// TwinCAT 3 PLC project ModbusExt2
// Title: ModbusExt2
// Company: Beckhoff Automation
// ProjectVersion: 0.1.0.0
// ProgramVersion: 3.1.4026.27
// libraries:
//   Tc2_SerialCom, * (Beckhoff Automation GmbH)
//   Tc2_Standard, * (Beckhoff Automation GmbH)
//   Tc2_System, * (Beckhoff Automation GmbH)
//   Tc2_TcpIp, * (Beckhoff Automation GmbH)
//   Tc2_Utilities, * (Beckhoff Automation GmbH)
// project tree:
//   DUTs/ E_MbAddressing.TcDUT, E_MbDevState.TcDUT, E_MbErrorClass.TcDUT, E_MbLogWriterStep.TcDUT, E_MbOp.TcDUT, E_MbPoll.TcDUT, E_MbRegion.TcDUT, E_MbTcpConn.TcDUT, E_MbType.TcDUT, E_MbWordOrder.TcDUT, E_MbXferState.TcDUT, ST_MbBlock.TcDUT, ST_MbLog.TcDUT, ST_MbLogEntry.TcDUT, ST_MbParseResult.TcDUT, ST_MbPoint.TcDUT, ST_MbPointState.TcDUT, ST_MbProbe.TcDUT, ST_MbProfile.TcDUT, U_MbConv.TcDUT
//   GVLs/ GVL_MbConst.TcGVL, GVL_MbParam.TcGVL
//   POUs/Codec/ F_MbCrc16.TcPOU, F_MbDecode.TcPOU, F_MbEncode.TcPOU, F_MbExpectedResponseLength.TcPOU, F_MbBuildRequest.TcPOU, F_MbMemCpy.TcPOU, F_MbMemSet.TcPOU, F_MbParseResponse.TcPOU, F_MbRound.TcPOU, F_MbTimeToFt.TcPOU
//   POUs/Device/ FB_ModbusDevice.TcPOU
//   POUs/Log/ FB_MbLogExport.TcPOU, FB_MbLogWriter.TcPOU, F_MbLogEntryToCsv.TcPOU
//   POUs/Profiles/ FB_Mb_CorrAll.TcPOU
//   POUs/Transport/ FB_MbTransportMock.TcPOU, FB_MbTransportRtu.TcPOU, FB_MbTransportTcp.TcPOU, I_MbTransport.TcIO
// real-time tasks:
//   TASK PlcTask1: cycle T#10ms, priority 21, ADS port 351
//   TASK PlcTask: cycle T#10ms, priority 20, ADS port 350

// ---- DUTs/E_MbAddressing.TcDUT
{attribute 'qualified_only'}
{attribute 'strict'}
TYPE E_MbAddressing :
(
	Modicon := 0,
	Offset0,
	Offset1
);
END_TYPE

// ---- DUTs/E_MbDevState.TcDUT
{attribute 'qualified_only'}
{attribute 'strict'}
TYPE E_MbDevState :
(
	Idle := 0,
	Acquire,
	Wait,
	Cooldown
);
END_TYPE

// ---- DUTs/E_MbErrorClass.TcDUT
{attribute 'qualified_only'}
{attribute 'strict'}
{attribute 'to_string'}
TYPE E_MbErrorClass :
(
	None := 0,
	Timeout,
	Crc,
	Exception,
	Transport,
	Config,
	Truncated,
	Malformed,
	StillFailing,
	Recovered
);
END_TYPE

// ---- DUTs/E_MbLogWriterStep.TcDUT
{attribute 'qualified_only'}
{attribute 'strict'}
TYPE E_MbLogWriterStep :
(
	Idle := 0,
	MkDir,
	MkDirWait,
	Open,
	OpenWait,
	SeekWait,
	TellWait,
	PutWait,
	CloseWait,
	DeleteWait,
	RenameWait
);
END_TYPE

// ---- DUTs/E_MbOp.TcDUT
{attribute 'qualified_only'}
{attribute 'strict'}
{attribute 'to_string'}
TYPE E_MbOp :
(
	Read := 0,
	Write
);
END_TYPE

// ---- DUTs/E_MbPoll.TcDUT
{attribute 'qualified_only'}
{attribute 'strict'}
TYPE E_MbPoll :
(
	Fast := 0,
	Slow,
	Off
);
END_TYPE

// ---- DUTs/E_MbRegion.TcDUT
{attribute 'qualified_only'}
{attribute 'strict'}
{attribute 'to_string'}
TYPE E_MbRegion :
(
	Auto := 0,
	Coil,
	DiscreteInput,
	InputRegister,
	HoldingRegister
);
END_TYPE

// ---- DUTs/E_MbTcpConn.TcDUT
{attribute 'qualified_only'}
{attribute 'strict'}
TYPE E_MbTcpConn :
(
	Init := 0,
	CloseAllWait,
	Disconnected,
	Connecting,
	Connected,
	Closing,
	ClosingWait
);
END_TYPE

// ---- DUTs/E_MbType.TcDUT
{attribute 'qualified_only'}
{attribute 'strict'}
TYPE E_MbType :
(
	Auto := 0,
	Boolean,
	Int16,
	UInt16,
	Int32,
	UInt32,
	Real32,
	Int64,
	UInt64,
	Real64,
	RegisterBit,
	Text,
	Raw
);
END_TYPE

// ---- DUTs/E_MbWordOrder.TcDUT
{attribute 'qualified_only'}
{attribute 'strict'}
TYPE E_MbWordOrder :
(
	Inherit := 0,
	ABCD,
	CDAB,
	BADC,
	DCBA
);
END_TYPE

// ---- DUTs/E_MbXferState.TcDUT
{attribute 'qualified_only'}
{attribute 'strict'}
TYPE E_MbXferState :
(
	Idle := 0,
	Busy,
	Done,
	Timeout,
	Error
);
END_TYPE

// ---- DUTs/ST_MbBlock.TcDUT
TYPE ST_MbBlock :
STRUCT
	eRegion      : E_MbRegion;
	nOffset      : UINT;       // 0-based start address
	nCount       : UINT;       // Registers or coils
	nFc          : USINT;      // Read function code
	ePoll        : E_MbPoll;
	nSortedFirst : UINT;       // Index range into FB_ModbusDevice.aSorted
	nSortedCount : UINT;
	tLastPoll    : ULINT;      // FILETIME of last completed poll (Slow scheduling)
	nConsecFail  : UINT;
END_STRUCT
END_TYPE

// ---- DUTs/ST_MbLog.TcDUT
TYPE ST_MbLog :
STRUCT
	aEntries     : ARRAY[0..GVL_MbParam.MB_LOG_SIZE-1] OF ST_MbLogEntry;
	nHead        : UINT;                             // Next write index
	nCount       : UINT;                             // Valid entries, <= MB_LOG_SIZE
	nTotalErrors : UDINT;
	nDropped     : UDINT;                            // Entries overwritten by ring wrap
	nSeq         : UDINT;                            // Entries ever written; the file writer's cursor
END_STRUCT
END_TYPE

// ---- DUTs/ST_MbLogEntry.TcDUT
TYPE ST_MbLogEntry :
STRUCT
	tTime    : ULINT;                                // FILETIME (100 ns, UTC)
	sName    : STRING(GVL_MbParam.MB_NAME_LEN);
	nUnitId  : USINT;
	eRegion  : E_MbRegion;
	nAddr    : UDINT;                                // As entered in the profile
	nFc      : BYTE;
	eOp      : E_MbOp;
	eClass   : E_MbErrorClass;
	nExcCode : BYTE;
	nRetries : USINT;
	nRepeat  : UDINT;                                // StillFailing: occurrences since first failure
END_STRUCT
END_TYPE

// ---- DUTs/ST_MbParseResult.TcDUT
TYPE ST_MbParseResult :
STRUCT
	bOk         : BOOL;             // Valid non-exception response matching the request
	bException  : BOOL;
	nExcCode    : BYTE;             // Modbus exception code when bException
	eClass      : E_MbErrorClass;   // None | Exception | Truncated | Malformed
	nByteCount  : UINT;             // Data bytes (FC 1..4)
	nDataOffset : UINT;             // Index of first data byte within the PDU (FC 1..4)
END_STRUCT
END_TYPE

// ---- DUTs/ST_MbPoint.TcDUT
TYPE ST_MbPoint :
STRUCT
	// ---- Profile fills these ----
	nAddr         : UDINT;                                   // Address as printed in the device manual (see E_MbAddressing)
	eType         : E_MbType     := E_MbType.Auto;           // Auto: Boolean for bit regions, UInt16 for registers
	eRegion       : E_MbRegion   := E_MbRegion.Auto;         // Auto: derived from nAddr (Modicon); required for Offset0/Offset1
	eWordOrder    : E_MbWordOrder := E_MbWordOrder.Inherit;  // Inherit from Profile()
	fRawMin       : LREAL;                                   // Scaling active iff fRawMin <> fRawMax
	fRawMax       : LREAL;
	fEngMin       : LREAL;
	fEngMax       : LREAL;
	fGain         : LREAL;                                   // Alternative scaling: eng = raw * fGain + fOffset. Active iff fGain <> 0
	fOffset       : LREAL;
	ePoll         : E_MbPoll     := E_MbPoll.Fast;
	bUseFailValue : BOOL;                                    // TRUE: fValue := fFailValue after retries exhausted
	fFailValue    : LREAL;
	nRegs         : UINT;                                    // Text/Raw only: registers to read
	nBit          : USINT;                                   // RegisterBit only: 0..15

	// ---- Library fills these ----
	fValue        : LREAL;                                   // Scaled value (numeric, Boolean, RegisterBit)
	sValue        : STRING(GVL_MbParam.MB_STR_LEN);          // Text
	aRaw          : ARRAY[0..GVL_MbParam.MB_RAW_WORDS-1] OF WORD;  // Raw, and raw words of every read
	bValid        : BOOL;
	tLastGood     : ULINT;                                   // FILETIME (100 ns, UTC) of last good read
	nFailCount    : UDINT;
	bProbe        : BOOL;                                    // User sets; cleared after stProbe is filled

	// ---- Write handshake ----
	fWriteValue   : LREAL;
	bWriteReq     : BOOL;
	bWriteBusy    : BOOL;
	bWriteDone    : BOOL;
	bWriteErr     : BOOL;

	// ---- Internal ----
	wMagic        : WORD := 16#4D50;
	nIndex        : UINT;
END_STRUCT
END_TYPE

// ---- DUTs/ST_MbPointState.TcDUT
TYPE ST_MbPointState :
STRUCT
	pPoint      : POINTER TO ST_MbPoint;   // Re-established in FB_reinit
	sName       : STRING(GVL_MbParam.MB_NAME_LEN);
	eRegion     : E_MbRegion;              // Resolved
	nOffset     : UINT;                    // Resolved 0-based address
	nCount      : UINT;                    // Registers or coils occupied
	eType       : E_MbType;                // Resolved (Auto replaced)
	eWordOrder  : E_MbWordOrder;           // Resolved (Inherit replaced)
	nReadFc     : USINT;
	nWriteFc    : USINT;                   // 0 = not writable
	nBlock      : UINT;                    // Owning read block; MB_MAX_BLOCKS = none (Poll Off)
	bFailing    : BOOL;
	nRepeat     : UDINT;
	tLastLog    : ULINT;
	eLastClass  : E_MbErrorClass;
	nLastExc    : BYTE;
	nWriteState : USINT;                   // 0 idle, 1 queued, 2 in flight
	aWriteData  : ARRAY[0..7] OF BYTE;
	cbWriteData : USINT;
	nWriteQty   : UINT;
END_STRUCT
END_TYPE

// ---- DUTs/ST_MbProbe.TcDUT
TYPE ST_MbProbe :
STRUCT
	sName        : STRING(GVL_MbParam.MB_NAME_LEN);
	nAddr        : UDINT;
	aRaw         : ARRAY[0..3] OF WORD;              // First four registers as received
	nInt16       : INT;
	nUInt16      : UINT;
	nInt32_ABCD  : DINT;
	nInt32_CDAB  : DINT;
	nInt32_BADC  : DINT;
	nInt32_DCBA  : DINT;
	nUInt32_ABCD : UDINT;
	nUInt32_CDAB : UDINT;
	nUInt32_BADC : UDINT;
	nUInt32_DCBA : UDINT;
	fReal32_ABCD : REAL;
	fReal32_CDAB : REAL;
	fReal32_BADC : REAL;
	fReal32_DCBA : REAL;
END_STRUCT
END_TYPE

// ---- DUTs/ST_MbProfile.TcDUT
TYPE ST_MbProfile :
STRUCT
	sModel          : STRING(GVL_MbParam.MB_NAME_LEN);
	eWordOrder      : E_MbWordOrder  := E_MbWordOrder.ABCD;
	eAddressing     : E_MbAddressing := E_MbAddressing.Modicon;
	nMaxRegsPerRead : UINT := GVL_MbConst.MAX_READ_REGS;
	nMaxGap         : UINT := 8;
	bFc6Only        : BOOL;
	bFc16Only       : BOOL;
	bStringByteSwap : BOOL;
	tSlowPoll       : TIME := T#5S;
END_STRUCT
END_TYPE

// ---- DUTs/U_MbConv.TcDUT
TYPE U_MbConv :
UNION
	lw : LWORD;
	dw : DWORD;
	w  : WORD;
	i  : INT;
	di : DINT;
	li : LINT;
	fR : REAL;
	fL : LREAL;
END_UNION
END_TYPE

// ---- GVLs/GVL_MbConst.TcGVL
{attribute 'qualified_only'}
VAR_GLOBAL CONSTANT
	FC_READ_COILS      : USINT := 1;
	FC_READ_DISCRETE   : USINT := 2;
	FC_READ_HOLDING    : USINT := 3;
	FC_READ_INPUT      : USINT := 4;
	FC_WRITE_COIL      : USINT := 5;
	FC_WRITE_REGISTER  : USINT := 6;
	FC_WRITE_COILS     : USINT := 15;
	FC_WRITE_REGISTERS : USINT := 16;
	EXC_FLAG           : BYTE  := 16#80;
	MAX_READ_REGS      : UINT  := 125;
	MAX_WRITE_REGS     : UINT  := 123;
	MAX_READ_COILS     : UINT  := 2000;
	MAX_WRITE_COILS    : UINT  := 1968;
	CFG_TOO_MANY_POINTS : BYTE := 1;
	CFG_NO_POINTS       : BYTE := 2;
	CFG_BAD_MAGIC       : BYTE := 3;
	CFG_EMPTY_NAME      : BYTE := 4;
	CFG_DUP_NAME        : BYTE := 5;
	CFG_BAD_ADDRESS     : BYTE := 6;
	CFG_REGION_REQUIRED : BYTE := 7;
	CFG_REGION_MISMATCH : BYTE := 8;
	CFG_BAD_TYPE        : BYTE := 9;
	CFG_BAD_REGS        : BYTE := 10;
	CFG_BAD_BIT         : BYTE := 11;
	CFG_BAD_SCALING     : BYTE := 12;
	CFG_OVERLAP         : BYTE := 13;
	CFG_TOO_MANY_BLOCKS : BYTE := 14;
	CFG_BAD_FAILVALUE   : BYTE := 15;
	CFG_NO_TRANSPORT    : BYTE := 16;
	CFG_NOT_WRITABLE    : BYTE := 17;
	CFG_WRITE_RANGE     : BYTE := 18;
END_VAR

// ---- GVLs/GVL_MbParam.TcGVL
{attribute 'qualified_only'}
VAR_GLOBAL CONSTANT
	MB_MAX_POINTS                : UINT := 256;
	MB_MAX_BLOCKS                : UINT := 64;
	MB_LOG_SIZE                  : UINT := 100;
	MB_STR_LEN                   : UINT := 32;
	MB_RAW_WORDS                 : UINT := 8;
	MB_NAME_LEN                  : UINT := 32;
	MB_MAX_DEVICES_PER_TRANSPORT : UINT := 32;
	MB_ADU_SIZE                  : UINT := 260;
	MB_LOG_REPEAT_INTERVAL       : TIME := T#5M;
	MB_OFFLINE_RETRY             : TIME := T#5S;
	MB_LOG_DIR                   : STRING(255) := 'C:\ModbusExt\Logs\';
	MB_LOG_FILE_MAX_BYTES        : UDINT := 2000000;   // Rotate to <name>.1.csv above this
	MB_LOG_FILE_BATCH            : USINT := 20;        // Entries per open/close
	MB_LOG_FILE_RETRY            : TIME  := T#10S;     // Backoff after a file error
END_VAR

// ---- POUs/Transport/I_MbTransport.TcIO
INTERFACE I_MbTransport

METHOD Abort
VAR_INPUT
	nUnitId : USINT;
END_VAR
END_METHOD

METHOD Acquire : BOOL
VAR_INPUT
	nUnitId : USINT;   // Caller's unit ID doubles as the owner key. TRUE = you hold the bus.
END_VAR
END_METHOD

PROPERTY bReady : BOOL
GET
END_GET
END_PROPERTY

PROPERTY cbResponsePdu : UINT
GET
END_GET
END_PROPERTY

PROPERTY eLastError : E_MbErrorClass
GET
END_GET
END_PROPERTY

METHOD Poll : E_MbXferState
END_METHOD

PROPERTY pResponsePdu : POINTER TO BYTE
GET
END_GET
END_PROPERTY

METHOD Release
VAR_INPUT
	nUnitId : USINT;
END_VAR
END_METHOD

METHOD Send : BOOL
VAR_INPUT
	nUnitId         : USINT;
	pPdu            : POINTER TO BYTE;
	cbPdu           : UINT;
	nExpectedPduLen : UINT;   // From F_MbExpectedResponseLength; RTU uses it to detect end of frame
	tTimeout        : TIME;
END_VAR
END_METHOD

END_INTERFACE

// ---- POUs/Codec/F_MbCrc16.TcPOU
FUNCTION F_MbCrc16 : WORD
VAR_INPUT
	pData : POINTER TO BYTE;
	cbLen : UDINT;
END_VAR
VAR
	i    : UDINT;
	j    : USINT;
	wCrc : WORD;
END_VAR

// Modbus RTU CRC-16: poly 16#A001 (reflected 16#8005), init 16#FFFF.
// Wire order is low byte first: CRC 16#8776 is sent as 76 87.
F_MbCrc16 := 16#FFFF;
IF pData = 0 OR cbLen = 0 THEN
	RETURN;
END_IF

wCrc := 16#FFFF;
FOR i := 0 TO cbLen - 1 DO
	wCrc := wCrc XOR BYTE_TO_WORD(pData[i]);
	FOR j := 1 TO 8 DO
		IF (wCrc AND 16#0001) <> 0 THEN
			wCrc := SHR(wCrc, 1) XOR 16#A001;
		ELSE
			wCrc := SHR(wCrc, 1);
		END_IF
	END_FOR
END_FOR
F_MbCrc16 := wCrc;

END_FUNCTION

// ---- POUs/Codec/F_MbDecode.TcPOU
FUNCTION F_MbDecode : LREAL
VAR_INPUT
	pSrc       : POINTER TO BYTE;   // First data byte; registers are big-endian on the wire
	nWords     : UINT;              // 1, 2 or 4
	eType      : E_MbType;
	eWordOrder : E_MbWordOrder;
	nBit       : USINT;             // RegisterBit only
END_VAR
VAR
	k, src     : UINT;
	w          : WORD;
	bByteSwap  : BOOL;
	bWordRev   : BOOL;
	u          : U_MbConv;
END_VAR

F_MbDecode := 0;
IF pSrc = 0 OR nWords < 1 OR nWords > 4 THEN
	RETURN;
END_IF

bByteSwap := (eWordOrder = E_MbWordOrder.BADC) OR (eWordOrder = E_MbWordOrder.DCBA);
bWordRev  := (eWordOrder = E_MbWordOrder.CDAB) OR (eWordOrder = E_MbWordOrder.DCBA);

// Assemble most-significant word first
u.lw := 0;
FOR k := 0 TO nWords - 1 DO
	src := SEL(bWordRev, k, nWords - 1 - k);
	IF bByteSwap THEN
		w := SHL(BYTE_TO_WORD(pSrc[2 * src + 1]), 8) OR BYTE_TO_WORD(pSrc[2 * src]);
	ELSE
		w := SHL(BYTE_TO_WORD(pSrc[2 * src]), 8) OR BYTE_TO_WORD(pSrc[2 * src + 1]);
	END_IF
	u.lw := SHL(u.lw, 16) OR WORD_TO_LWORD(w);
END_FOR

CASE eType OF
	E_MbType.Boolean:     F_MbDecode := SEL(u.w <> 0, 0.0, 1.0);
	E_MbType.Int16:       F_MbDecode := INT_TO_LREAL(u.i);
	E_MbType.UInt16:      F_MbDecode := UINT_TO_LREAL(WORD_TO_UINT(u.w));
	E_MbType.Int32:       F_MbDecode := DINT_TO_LREAL(u.di);
	E_MbType.UInt32:      F_MbDecode := UDINT_TO_LREAL(DWORD_TO_UDINT(u.dw));
	E_MbType.Real32:      F_MbDecode := REAL_TO_LREAL(u.fR);
	E_MbType.Int64:       F_MbDecode := LINT_TO_LREAL(u.li);
	E_MbType.UInt64:      F_MbDecode := ULINT_TO_LREAL(LWORD_TO_ULINT(u.lw));
	E_MbType.Real64:      F_MbDecode := u.fL;
	E_MbType.RegisterBit: F_MbDecode := SEL((u.w AND SHL(WORD#1, nBit)) <> 0, 0.0, 1.0);
END_CASE

END_FUNCTION

// ---- POUs/Codec/F_MbEncode.TcPOU
FUNCTION F_MbEncode : BOOL
VAR_INPUT
	fValue     : LREAL;
	eType      : E_MbType;
	eWordOrder : E_MbWordOrder;
	pDst       : POINTER TO BYTE;   // 2*nWords bytes, written big-endian in the configured order
	nWords     : UINT;
END_VAR
VAR
	u          : U_MbConv;
	k, dst     : UINT;
	w          : WORD;
	fR         : LREAL;
	bByteSwap  : BOOL;
	bWordRev   : BOOL;
END_VAR

// FALSE = value out of range for the target type
F_MbEncode := FALSE;
IF pDst = 0 OR nWords < 1 OR nWords > 4 THEN
	RETURN;
END_IF

u.lw := 0;
fR   := F_MbRound(fValue);
CASE eType OF
	E_MbType.Int16:
		IF fR < -32768.0 OR fR > 32767.0 THEN RETURN; END_IF
		u.i := LREAL_TO_INT(fR);
	E_MbType.UInt16:
		IF fR < 0.0 OR fR > 65535.0 THEN RETURN; END_IF
		u.w := UINT_TO_WORD(LREAL_TO_UINT(fR));
	E_MbType.Int32:
		IF fR < -2147483648.0 OR fR > 2147483647.0 THEN RETURN; END_IF
		u.di := LREAL_TO_DINT(fR);
	E_MbType.UInt32:
		IF fR < 0.0 OR fR > 4294967295.0 THEN RETURN; END_IF
		u.dw := UDINT_TO_DWORD(LREAL_TO_UDINT(fR));
	E_MbType.Int64:
		u.li := LREAL_TO_LINT(fR);
	E_MbType.UInt64:
		IF fR < 0.0 THEN RETURN; END_IF
		u.lw := ULINT_TO_LWORD(LREAL_TO_ULINT(fR));
	E_MbType.Real32:
		IF ABS(fValue) > 3.4028234E38 THEN RETURN; END_IF
		u.fR := LREAL_TO_REAL(fValue);
	E_MbType.Real64:
		u.fL := fValue;
ELSE
	RETURN;
END_CASE

bByteSwap := (eWordOrder = E_MbWordOrder.BADC) OR (eWordOrder = E_MbWordOrder.DCBA);
bWordRev  := (eWordOrder = E_MbWordOrder.CDAB) OR (eWordOrder = E_MbWordOrder.DCBA);
FOR k := 0 TO nWords - 1 DO
	w   := LWORD_TO_WORD(SHR(u.lw, 16 * (nWords - 1 - k)));   // k-th word, most significant first
	dst := SEL(bWordRev, k, nWords - 1 - k);
	IF bByteSwap THEN
		pDst[2 * dst]     := WORD_TO_BYTE(w);
		pDst[2 * dst + 1] := WORD_TO_BYTE(SHR(w, 8));
	ELSE
		pDst[2 * dst]     := WORD_TO_BYTE(SHR(w, 8));
		pDst[2 * dst + 1] := WORD_TO_BYTE(w);
	END_IF
END_FOR
F_MbEncode := TRUE;

END_FUNCTION

// ---- POUs/Codec/F_MbRound.TcPOU
FUNCTION F_MbRound : LREAL
VAR_INPUT
	f  : LREAL;
END_VAR
VAR
	fR : LREAL;
END_VAR

// Round half away from zero. Exact below 2^31; larger magnitudes pass through.
IF f >= 0 THEN
	fR := f + 0.5;
ELSE
	fR := f - 0.5;
END_IF
IF ABS(fR) < 2147483647.0 THEN
	F_MbRound := DINT_TO_LREAL(TRUNC(fR));
ELSE
	F_MbRound := f;
END_IF

END_FUNCTION

// ---- POUs/Codec/F_MbExpectedResponseLength.TcPOU
FUNCTION F_MbExpectedResponseLength : UINT
VAR_INPUT
	nFc  : USINT;
	nQty : UINT;
END_VAR

// PDU bytes of a normal response (no unit ID, CRC or MBAP). 0 = unsupported FC.
// An exception response is always 2 PDU bytes; transports check for that separately.
CASE nFc OF
	GVL_MbConst.FC_READ_COILS, GVL_MbConst.FC_READ_DISCRETE:
		F_MbExpectedResponseLength := 2 + (nQty + 7) / 8;
	GVL_MbConst.FC_READ_HOLDING, GVL_MbConst.FC_READ_INPUT:
		F_MbExpectedResponseLength := 2 + 2 * nQty;
	GVL_MbConst.FC_WRITE_COIL, GVL_MbConst.FC_WRITE_REGISTER,
	GVL_MbConst.FC_WRITE_COILS, GVL_MbConst.FC_WRITE_REGISTERS:
		F_MbExpectedResponseLength := 5;
ELSE
	F_MbExpectedResponseLength := 0;
END_CASE

END_FUNCTION

// ---- POUs/Codec/F_MbBuildRequest.TcPOU
FUNCTION F_MbBuildRequest : UINT
VAR_INPUT
	nFc      : USINT;             // GVL_MbConst.FC_*
	nOffset  : UINT;              // 0-based PDU address
	nQty     : UINT;              // FC 1,2,3,4,15,16. Ignored for FC 5,6
	pData    : POINTER TO BYTE;   // FC5/6: 2 bytes big-endian. FC15: packed coils. FC16: registers big-endian
	cbData   : UINT;              // Payload length
	pPdu     : POINTER TO BYTE;   // Output buffer
	cbPduMax : UINT;              // Output buffer size
END_VAR
VAR
	nLen     : UINT;
	nByteCnt : UINT;
END_VAR

// Returns the PDU length written to pPdu, or 0 if the request is invalid.
F_MbBuildRequest := 0;
IF pPdu = 0 OR cbPduMax < 5 THEN
	RETURN;
END_IF

pPdu[0] := USINT_TO_BYTE(nFc);
pPdu[1] := UINT_TO_BYTE(SHR(nOffset, 8));
pPdu[2] := UINT_TO_BYTE(nOffset);

CASE nFc OF
	GVL_MbConst.FC_READ_COILS, GVL_MbConst.FC_READ_DISCRETE:
		IF nQty < 1 OR nQty > GVL_MbConst.MAX_READ_COILS THEN
			RETURN;
		END_IF
		pPdu[3] := UINT_TO_BYTE(SHR(nQty, 8));
		pPdu[4] := UINT_TO_BYTE(nQty);
		nLen := 5;

	GVL_MbConst.FC_READ_HOLDING, GVL_MbConst.FC_READ_INPUT:
		IF nQty < 1 OR nQty > GVL_MbConst.MAX_READ_REGS THEN
			RETURN;
		END_IF
		pPdu[3] := UINT_TO_BYTE(SHR(nQty, 8));
		pPdu[4] := UINT_TO_BYTE(nQty);
		nLen := 5;

	GVL_MbConst.FC_WRITE_COIL, GVL_MbConst.FC_WRITE_REGISTER:
		IF pData = 0 OR cbData <> 2 THEN
			RETURN;
		END_IF
		pPdu[3] := pData[0];
		pPdu[4] := pData[1];
		nLen := 5;

	GVL_MbConst.FC_WRITE_COILS:
		IF nQty < 1 OR nQty > GVL_MbConst.MAX_WRITE_COILS THEN
			RETURN;
		END_IF
		nByteCnt := (nQty + 7) / 8;
		IF pData = 0 OR cbData <> nByteCnt OR cbPduMax < 6 + nByteCnt THEN
			RETURN;
		END_IF
		pPdu[3] := UINT_TO_BYTE(SHR(nQty, 8));
		pPdu[4] := UINT_TO_BYTE(nQty);
		pPdu[5] := UINT_TO_BYTE(nByteCnt);
		F_MbMemCpy(pPdu + 6, pData, nByteCnt);
		nLen := 6 + nByteCnt;

	GVL_MbConst.FC_WRITE_REGISTERS:
		IF nQty < 1 OR nQty > GVL_MbConst.MAX_WRITE_REGS THEN
			RETURN;
		END_IF
		nByteCnt := 2 * nQty;
		IF pData = 0 OR cbData <> nByteCnt OR cbPduMax < 6 + nByteCnt THEN
			RETURN;
		END_IF
		pPdu[3] := UINT_TO_BYTE(SHR(nQty, 8));
		pPdu[4] := UINT_TO_BYTE(nQty);
		pPdu[5] := UINT_TO_BYTE(nByteCnt);
		F_MbMemCpy(pPdu + 6, pData, nByteCnt);
		nLen := 6 + nByteCnt;
ELSE
	RETURN;
END_CASE

F_MbBuildRequest := nLen;

END_FUNCTION

// ---- POUs/Codec/F_MbMemCpy.TcPOU
FUNCTION F_MbMemCpy : BOOL
VAR_INPUT
	pDst : POINTER TO BYTE;
	pSrc : POINTER TO BYTE;
	n    : UDINT;
END_VAR
VAR
	i    : UDINT;
END_VAR

// Forward copy: safe for overlapping ranges when pDst <= pSrc (all our moves go downward)
F_MbMemCpy := FALSE;
IF pDst = 0 OR pSrc = 0 THEN
	RETURN;
END_IF
IF n > 0 THEN
	FOR i := 0 TO n - 1 DO
		pDst[i] := pSrc[i];
	END_FOR
END_IF
F_MbMemCpy := TRUE;

END_FUNCTION

// ---- POUs/Codec/F_MbMemSet.TcPOU
FUNCTION F_MbMemSet : BOOL
VAR_INPUT
	pDst : POINTER TO BYTE;
	b    : BYTE;
	n    : UDINT;
END_VAR
VAR
	i    : UDINT;
END_VAR

F_MbMemSet := FALSE;
IF pDst = 0 THEN
	RETURN;
END_IF
IF n > 0 THEN
	FOR i := 0 TO n - 1 DO
		pDst[i] := b;
	END_FOR
END_IF
F_MbMemSet := TRUE;

END_FUNCTION

// ---- POUs/Codec/F_MbParseResponse.TcPOU
FUNCTION F_MbParseResponse : BOOL
VAR_INPUT
	pPdu         : POINTER TO BYTE;   // Response PDU, starting at the function code
	cbPdu        : UINT;
	nFcExpected  : USINT;
	nQtyExpected : UINT;              // Quantity from the request (FC 1,2,3,4,15,16)
END_VAR
VAR_IN_OUT
	stResult     : ST_MbParseResult;
END_VAR
VAR
	nFc      : USINT;
	nByteCnt : UINT;
	nQtyEcho : UINT;
END_VAR

// Returns stResult.bOk. Never reads past cbPdu.
F_MbParseResponse    := FALSE;
stResult.bOk         := FALSE;
stResult.bException  := FALSE;
stResult.nExcCode    := 0;
stResult.eClass      := E_MbErrorClass.None;
stResult.nByteCount  := 0;
stResult.nDataOffset := 0;

IF pPdu = 0 OR cbPdu < 1 THEN
	stResult.eClass := E_MbErrorClass.Truncated;
	RETURN;
END_IF

// Exception response: (FC OR 16#80) followed by one code byte
IF pPdu[0] = (USINT_TO_BYTE(nFcExpected) OR GVL_MbConst.EXC_FLAG) THEN
	IF cbPdu < 2 THEN
		stResult.eClass := E_MbErrorClass.Truncated;
	ELSE
		stResult.bException := TRUE;
		stResult.nExcCode   := pPdu[1];
		stResult.eClass     := E_MbErrorClass.Exception;
	END_IF
	RETURN;
END_IF

nFc := BYTE_TO_USINT(pPdu[0]);
IF nFc <> nFcExpected THEN
	stResult.eClass := E_MbErrorClass.Malformed;
	RETURN;
END_IF

CASE nFc OF
	GVL_MbConst.FC_READ_COILS, GVL_MbConst.FC_READ_DISCRETE,
	GVL_MbConst.FC_READ_HOLDING, GVL_MbConst.FC_READ_INPUT:
		IF cbPdu < 2 THEN
			stResult.eClass := E_MbErrorClass.Truncated;
			RETURN;
		END_IF
		nByteCnt := BYTE_TO_UINT(pPdu[1]);
		IF nFc <= GVL_MbConst.FC_READ_DISCRETE THEN
			IF nByteCnt <> (nQtyExpected + 7) / 8 THEN
				stResult.eClass := E_MbErrorClass.Malformed;
				RETURN;
			END_IF
		ELSIF nByteCnt <> 2 * nQtyExpected THEN
			stResult.eClass := E_MbErrorClass.Malformed;
			RETURN;
		END_IF
		IF cbPdu < 2 + nByteCnt THEN
			stResult.eClass := E_MbErrorClass.Truncated;
			RETURN;
		END_IF
		stResult.nByteCount  := nByteCnt;
		stResult.nDataOffset := 2;
		stResult.bOk         := TRUE;

	GVL_MbConst.FC_WRITE_COIL, GVL_MbConst.FC_WRITE_REGISTER:
		IF cbPdu < 5 THEN
			stResult.eClass := E_MbErrorClass.Truncated;
			RETURN;
		END_IF
		stResult.bOk := TRUE;

	GVL_MbConst.FC_WRITE_COILS, GVL_MbConst.FC_WRITE_REGISTERS:
		IF cbPdu < 5 THEN
			stResult.eClass := E_MbErrorClass.Truncated;
			RETURN;
		END_IF
		nQtyEcho := SHL(BYTE_TO_UINT(pPdu[3]), 8) + BYTE_TO_UINT(pPdu[4]);
		IF nQtyEcho <> nQtyExpected THEN
			stResult.eClass := E_MbErrorClass.Malformed;
			RETURN;
		END_IF
		stResult.bOk := TRUE;
ELSE
	stResult.eClass := E_MbErrorClass.Malformed;
	RETURN;
END_CASE

F_MbParseResponse := stResult.bOk;

END_FUNCTION

// ---- POUs/Codec/F_MbTimeToFt.TcPOU
FUNCTION F_MbTimeToFt : ULINT
VAR_INPUT
	t : TIME;
END_VAR

// TIME (ms) -> FILETIME ticks (100 ns)
F_MbTimeToFt := UDINT_TO_ULINT(TIME_TO_UDINT(t)) * 10000;

END_FUNCTION

// ---- POUs/Device/FB_ModbusDevice.TcPOU
FUNCTION_BLOCK FB_ModbusDevice
VAR_INPUT
	itfTransport   : I_MbTransport;
	nUnitId        : USINT := 1;
	bEnable        : BOOL;
	tTimeout       : TIME  := T#500MS;
	nRetries       : USINT := 2;
	refLog         : REFERENCE TO ST_MbLog;   // Application-owned; may be PERSISTENT
	nOfflineAfter  : USINT := 3;        // Consecutive failed transactions before bOnline drops
	bLogToFile     : BOOL := TRUE;
	sLogDir        : STRING(255) := GVL_MbParam.MB_LOG_DIR;
	sLogName       : STRING(80);        // '' = <Model>_U<unit>
END_VAR
VAR_OUTPUT
	bOnline        : BOOL;
	bConfigError   : BOOL;
	nErrorCount    : UDINT;
	nTxCount       : UDINT;
	nRxCount       : UDINT;
	tLastRoundTrip : TIME;
	stLastError    : ST_MbLogEntry;
	stProbe        : ST_MbProbe;
	nPoints        : UINT;
	nBlocks        : UINT;
	nLogDropped    : UDINT;
	bLogFileError  : BOOL;
	nLogFileErrId  : UDINT;
	nLogWritten    : UDINT;
END_VAR
VAR
	stProfile      : ST_MbProfile;
	aState         : ARRAY[0..GVL_MbParam.MB_MAX_POINTS-1] OF ST_MbPointState;
	aSorted        : ARRAY[0..GVL_MbParam.MB_MAX_POINTS-1] OF UINT;   // Point indices ordered by region, offset
	aBlocks        : ARRAY[0..GVL_MbParam.MB_MAX_BLOCKS-1] OF ST_MbBlock;
	bAddOverflow   : BOOL;        // Add() called with the table full; reported by Init
	bInitDone      : BOOL;
	fbSysTime      : GETSYSTEMTIME;
	tNow           : ULINT;       // FILETIME, refreshed every cycle
	bNoTransportLogged : BOOL;
	eState         : E_MbDevState;
	nCurBlock      : UINT;
	nRotation      : UINT;
	nAttempt       : USINT;
	nConsecFailTx  : UINT;
	nDevRepeat     : UDINT;             // 0 = no device-level failure open
	tNextPoll      : ULINT;
	tTxStart       : ULINT;
	tLastDevLog    : ULINT;
	aPdu           : ARRAY[0..GVL_MbParam.MB_ADU_SIZE-1] OF BYTE;
	cbPdu          : UINT;
	nExpectedLen   : UINT;
	stParse        : ST_MbParseResult;
	nCurWrite      : UINT;
	bWriteTx       : BOOL;              // Current transaction is a write
	nRegCursor     : UINT;
	bRegChanged    : BOOL;
	stLog          : ST_MbLog;              // Internal ring, used when refLog is not bound
	pLog           : POINTER TO ST_MbLog;   // Active ring, refreshed every cycle
	fbLogWriter    : FB_MbLogWriter;
	sLogNameEff    : STRING(80);
END_VAR

fbSysTime();
tNow := SHL(DWORD_TO_ULINT(fbSysTime.timeHiDW), 32) + DWORD_TO_ULINT(fbSysTime.timeLoDW);

// Active ring: the caller's (persistent or merged) or our own. Refreshed every cycle.
IF __ISVALIDREF(refLog) THEN
	pLog := ADR(refLog);
ELSE
	pLog := ADR(stLog);
END_IF

// File writer: drains new entries in the background, even while disabled
IF LEN(sLogName) > 0 THEN
	sLogNameEff := sLogName;
ELSE
	sLogNameEff := CONCAT(CONCAT(stProfile.sModel, '_U'), USINT_TO_STRING(nUnitId));
END_IF
fbLogWriter(bEnable := bLogToFile, sDir := sLogDir, sName := sLogNameEff, pLog := pLog, tNow := tNow);
bLogFileError := fbLogWriter.bError;
nLogFileErrId := fbLogWriter.nErrId;
nLogWritten   := fbLogWriter.nWritten;

IF NOT bEnable THEN
	RETURN;
END_IF

// The profile registered its points just before SUPER^(); act only if the table changed
IF bRegChanged OR nRegCursor <> nPoints THEN
	nPoints     := nRegCursor;
	bRegChanged := FALSE;
	bInitDone   := FALSE;
END_IF

IF NOT bInitDone THEN
	Init();
END_IF
IF bConfigError THEN
	RETURN;
END_IF

IF itfTransport = 0 THEN
	IF NOT bNoTransportLogged THEN
		bNoTransportLogged := TRUE;
		WriteLog(nPoints, E_MbOp.Read, E_MbErrorClass.Config, 0, GVL_MbConst.CFG_NO_TRANSPORT, 0, 0);
	END_IF
	RETURN;
END_IF
bNoTransportLogged := FALSE;

ServiceWrites();
Scheduler();

METHOD PUBLIC AddPoint
VAR_IN_OUT
	stPoint : ST_MbPoint;
END_VAR
VAR_INPUT
	sName   : STRING;
END_VAR
IF nRegCursor >= GVL_MbParam.MB_MAX_POINTS THEN
	bAddOverflow := TRUE;
	RETURN;
END_IF
IF aState[nRegCursor].pPoint <> ADR(stPoint) OR aState[nRegCursor].sName <> sName THEN
	aState[nRegCursor].pPoint := ADR(stPoint);
	aState[nRegCursor].sName  := sName;
	bRegChanged := TRUE;
END_IF
stPoint.nIndex := nRegCursor;
nRegCursor     := nRegCursor + 1;
END_METHOD

METHOD PROTECTED BuildBlocks : BOOL
VAR
	k, idx    : UINT;
	nB        : UINT;        // Open block
	nBlockEnd : UDINT;       // Exclusive end offset of the open block
	nNewEnd   : UDINT;
	nMaxCount : UDINT;
	bBits     : BOOL;
	bOpen     : BOOL;
	ePoll     : E_MbPoll;
END_VAR
BuildBlocks := TRUE;
nBlocks := 0;
bOpen   := FALSE;
nB      := 0;

FOR k := 0 TO nPoints - 1 DO
	idx   := aSorted[k];
	ePoll := aState[idx].pPoint^.ePoll;
	IF ePoll = E_MbPoll.Off THEN
		aState[idx].nBlock := GVL_MbParam.MB_MAX_BLOCKS;
		CONTINUE;
	END_IF

	bBits := (aState[idx].eRegion = E_MbRegion.Coil) OR (aState[idx].eRegion = E_MbRegion.DiscreteInput);
	IF bBits THEN
		nMaxCount := GVL_MbConst.MAX_READ_COILS;
	ELSE
		nMaxCount := stProfile.nMaxRegsPerRead;
	END_IF
	nNewEnd := UINT_TO_UDINT(aState[idx].nOffset) + aState[idx].nCount;

	// Extend the open block: same region and poll class, gap small enough, span fits
	IF bOpen AND_THEN (aBlocks[nB].eRegion = aState[idx].eRegion AND aBlocks[nB].ePoll = ePoll)
	   AND_THEN (aState[idx].nOffset - nBlockEnd <= stProfile.nMaxGap)
	   AND_THEN (nNewEnd - aBlocks[nB].nOffset <= nMaxCount) THEN
		aBlocks[nB].nCount       := UDINT_TO_UINT(nNewEnd - aBlocks[nB].nOffset);
		aBlocks[nB].nSortedCount := aBlocks[nB].nSortedCount + 1;
		aState[idx].nBlock       := nB;
		nBlockEnd                := MAX(nBlockEnd, nNewEnd);
		CONTINUE;
	END_IF

	// Start a new block
	IF nBlocks >= GVL_MbParam.MB_MAX_BLOCKS THEN
		ConfigFail(idx, GVL_MbConst.CFG_TOO_MANY_BLOCKS);
		BuildBlocks := FALSE;
		RETURN;
	END_IF
	nB := nBlocks;
	aBlocks[nB].eRegion      := aState[idx].eRegion;
	aBlocks[nB].nOffset      := aState[idx].nOffset;
	aBlocks[nB].nCount       := aState[idx].nCount;
	aBlocks[nB].nFc          := aState[idx].nReadFc;
	aBlocks[nB].ePoll        := ePoll;
	aBlocks[nB].nSortedFirst := k;
	aBlocks[nB].nSortedCount := 1;
	aBlocks[nB].tLastPoll    := 0;
	aBlocks[nB].nConsecFail  := 0;
	aState[idx].nBlock       := nB;
	nBlockEnd                := nNewEnd;
	nBlocks                  := nBlocks + 1;
	bOpen                    := TRUE;
END_FOR
END_METHOD

METHOD PROTECTED ConfigFail
VAR_INPUT
	nPointIdx : UINT;   // >= nPoints means device-level
	nCode     : BYTE;   // GVL_MbConst.CFG_*
END_VAR
bConfigError := TRUE;
WriteLog(nPointIdx, E_MbOp.Read, E_MbErrorClass.Config, 0, nCode, 0, 0);
END_METHOD

METHOD PRIVATE DecodePoint
VAR_INPUT
	idx    : UINT;
	pSrc   : POINTER TO BYTE;   // First data byte of this point's registers
END_VAR
VAR
	pPt    : POINTER TO ST_MbPoint;
	nWords : UINT;
	k      : UINT;
	fRaw   : LREAL;
	pStr   : POINTER TO BYTE;
END_VAR
pPt    := aState[idx].pPoint;
nWords := aState[idx].nCount;

// Raw words as transmitted, capped at the buffer
FOR k := 0 TO MIN(nWords, GVL_MbParam.MB_RAW_WORDS) - 1 DO
	pPt^.aRaw[k] := SHL(BYTE_TO_WORD(pSrc[2 * k]), 8) OR BYTE_TO_WORD(pSrc[2 * k + 1]);
END_FOR

IF aState[idx].eType = E_MbType.Text THEN
	pStr := ADR(pPt^.sValue);
	FOR k := 0 TO nWords - 1 DO
		IF stProfile.bStringByteSwap THEN
			pStr[2 * k]     := pSrc[2 * k + 1];
			pStr[2 * k + 1] := pSrc[2 * k];
		ELSE
			pStr[2 * k]     := pSrc[2 * k];
			pStr[2 * k + 1] := pSrc[2 * k + 1];
		END_IF
	END_FOR
	pStr[2 * nWords] := 0;
	
ELSIF aState[idx].eType <> E_MbType.Raw THEN
	fRaw := F_MbDecode(pSrc, nWords, aState[idx].eType, aState[idx].eWordOrder, pPt^.nBit);
	IF pPt^.fGain <> 0 THEN
		pPt^.fValue := fRaw * pPt^.fGain + pPt^.fOffset;
	ELSIF pPt^.fRawMin <> pPt^.fRawMax THEN
		pPt^.fValue := pPt^.fEngMin + (fRaw - pPt^.fRawMin) * (pPt^.fEngMax - pPt^.fEngMin) / (pPt^.fRawMax - pPt^.fRawMin);
	ELSE
		pPt^.fValue := fRaw;
	END_IF
END_IF

IF pPt^.bProbe THEN
	FillProbe(idx, pSrc, nWords);
	pPt^.bProbe := FALSE;
END_IF
END_METHOD

METHOD PRIVATE EncodeWrite : BOOL
VAR_INPUT
	i    : UINT;
END_VAR
VAR
	pPt  : POINTER TO ST_MbPoint;
	fRaw : LREAL;
END_VAR
EncodeWrite := FALSE;
pPt := aState[i].pPoint;
IF pPt = 0 THEN
	RETURN;
END_IF

// Engineering -> raw (inverse of the read scaling)
fRaw := pPt^.fWriteValue;
IF pPt^.fGain <> 0 THEN
	fRaw := (fRaw - pPt^.fOffset) / pPt^.fGain;
ELSIF pPt^.fRawMin <> pPt^.fRawMax THEN
	fRaw := pPt^.fRawMin + (fRaw - pPt^.fEngMin) * (pPt^.fRawMax - pPt^.fRawMin) / (pPt^.fEngMax - pPt^.fEngMin);
END_IF

CASE aState[i].nWriteFc OF
	GVL_MbConst.FC_WRITE_COIL:
		aState[i].aWriteData[0] := SEL(fRaw <> 0, BYTE#16#00, BYTE#16#FF);
		aState[i].aWriteData[1] := BYTE#16#00;
		aState[i].cbWriteData   := 2;
		aState[i].nWriteQty     := 1;
	GVL_MbConst.FC_WRITE_COILS:
		aState[i].aWriteData[0] := SEL(fRaw <> 0, BYTE#16#00, BYTE#16#01);
		aState[i].cbWriteData   := 1;
		aState[i].nWriteQty     := 1;
	GVL_MbConst.FC_WRITE_REGISTER, GVL_MbConst.FC_WRITE_REGISTERS:
		aState[i].nWriteQty   := aState[i].nCount;
		aState[i].cbWriteData := UINT_TO_USINT(2 * aState[i].nCount);
		IF NOT F_MbEncode(fRaw, aState[i].eType, aState[i].eWordOrder, ADR(aState[i].aWriteData), aState[i].nCount) THEN
			RETURN;
		END_IF
ELSE
	RETURN;
END_CASE
EncodeWrite := TRUE;
END_METHOD

METHOD PRIVATE EndTransaction
VAR_INPUT
	bReachable : BOOL;
	eClass     : E_MbErrorClass;
	nExc       : BYTE;
END_VAR
itfTransport.Release(nUnitId);
eState := E_MbDevState.Cooldown;

IF bReachable THEN
	nConsecFailTx := 0;
	IF NOT bOnline THEN
		bOnline := TRUE;
		IF nDevRepeat > 0 THEN
			WriteLog(nPoints, E_MbOp.Read, E_MbErrorClass.Recovered, 0, 0, 0, nDevRepeat);
		END_IF
		nDevRepeat := 0;
	END_IF
	RETURN;
END_IF

nConsecFailTx := nConsecFailTx + 1;
IF bOnline AND nConsecFailTx < nOfflineAfter THEN
	RETURN;                                     // Still online; FailBlock logged the block
END_IF

bOnline := FALSE;
IF nDevRepeat = 0 THEN
	nDevRepeat  := 1;
	tLastDevLog := tNow;
	WriteLog(nPoints, E_MbOp.Read, eClass, 0, nExc, nRetries, 1);
ELSE
	nDevRepeat := nDevRepeat + 1;
	IF tNow - tLastDevLog >= F_MbTimeToFt(GVL_MbParam.MB_LOG_REPEAT_INTERVAL) THEN
		tLastDevLog := tNow;
		WriteLog(nPoints, E_MbOp.Read, E_MbErrorClass.StillFailing, 0, nExc, nRetries, nDevRepeat);
	END_IF
END_IF
tNextPoll := tNow + F_MbTimeToFt(GVL_MbParam.MB_OFFLINE_RETRY);
END_METHOD

METHOD PRIVATE FailBlock
VAR_INPUT
	eClass : E_MbErrorClass;
	nExc   : BYTE;
END_VAR
VAR
	k, idx, nFirst : UINT;
	pPt            : POINTER TO ST_MbPoint;
END_VAR
FOR k := 0 TO aBlocks[nCurBlock].nSortedCount - 1 DO
	idx := aSorted[aBlocks[nCurBlock].nSortedFirst + k];
	pPt := aState[idx].pPoint;
	IF pPt = 0 THEN
		CONTINUE;
	END_IF
	pPt^.bValid     := FALSE;
	pPt^.nFailCount := pPt^.nFailCount + 1;
	IF pPt^.bUseFailValue THEN
		pPt^.fValue := pPt^.fFailValue;
	END_IF
END_FOR
aBlocks[nCurBlock].nConsecFail := aBlocks[nCurBlock].nConsecFail + 1;
aBlocks[nCurBlock].tLastPoll   := tNow;

// One flood-controlled entry per block, keyed on its first point. Suppressed while offline.
nFirst := aSorted[aBlocks[nCurBlock].nSortedFirst];
aState[nFirst].eLastClass := eClass;
aState[nFirst].nLastExc   := nExc;
IF NOT aState[nFirst].bFailing THEN
	aState[nFirst].bFailing := TRUE;
	aState[nFirst].nRepeat  := 1;
	aState[nFirst].tLastLog := tNow;
	IF bOnline THEN
		WriteLog(nFirst, E_MbOp.Read, eClass, aBlocks[nCurBlock].nFc, nExc, nAttempt, 1);
	END_IF
ELSE
	aState[nFirst].nRepeat := aState[nFirst].nRepeat + 1;
	IF bOnline AND tNow - aState[nFirst].tLastLog >= F_MbTimeToFt(GVL_MbParam.MB_LOG_REPEAT_INTERVAL) THEN
		aState[nFirst].tLastLog := tNow;
		WriteLog(nFirst, E_MbOp.Read, E_MbErrorClass.StillFailing, aBlocks[nCurBlock].nFc, nExc, nAttempt, aState[nFirst].nRepeat);
	END_IF
END_IF
END_METHOD

METHOD PRIVATE FillProbe
VAR_INPUT
	idx     : UINT;
	pSrc    : POINTER TO BYTE;
	nWords  : UINT;
END_VAR
VAR
	k       : UINT;
	stEmpty : ST_MbProbe;
END_VAR
stProbe       := stEmpty;
stProbe.sName := aState[idx].sName;
stProbe.nAddr := aState[idx].pPoint^.nAddr;
FOR k := 0 TO 3 DO
	IF k < nWords THEN
		stProbe.aRaw[k] := SHL(BYTE_TO_WORD(pSrc[2 * k]), 8) OR BYTE_TO_WORD(pSrc[2 * k + 1]);
	END_IF
END_FOR
stProbe.nInt16  := LREAL_TO_INT(F_MbDecode(pSrc, 1, E_MbType.Int16, E_MbWordOrder.ABCD, 0));
stProbe.nUInt16 := LREAL_TO_UINT(F_MbDecode(pSrc, 1, E_MbType.UInt16, E_MbWordOrder.ABCD, 0));
IF nWords >= 2 THEN
	stProbe.nInt32_ABCD  := LREAL_TO_DINT(F_MbDecode(pSrc, 2, E_MbType.Int32, E_MbWordOrder.ABCD, 0));
	stProbe.nInt32_CDAB  := LREAL_TO_DINT(F_MbDecode(pSrc, 2, E_MbType.Int32, E_MbWordOrder.CDAB, 0));
	stProbe.nInt32_BADC  := LREAL_TO_DINT(F_MbDecode(pSrc, 2, E_MbType.Int32, E_MbWordOrder.BADC, 0));
	stProbe.nInt32_DCBA  := LREAL_TO_DINT(F_MbDecode(pSrc, 2, E_MbType.Int32, E_MbWordOrder.DCBA, 0));
	stProbe.nUInt32_ABCD := LREAL_TO_UDINT(F_MbDecode(pSrc, 2, E_MbType.UInt32, E_MbWordOrder.ABCD, 0));
	stProbe.nUInt32_CDAB := LREAL_TO_UDINT(F_MbDecode(pSrc, 2, E_MbType.UInt32, E_MbWordOrder.CDAB, 0));
	stProbe.nUInt32_BADC := LREAL_TO_UDINT(F_MbDecode(pSrc, 2, E_MbType.UInt32, E_MbWordOrder.BADC, 0));
	stProbe.nUInt32_DCBA := LREAL_TO_UDINT(F_MbDecode(pSrc, 2, E_MbType.UInt32, E_MbWordOrder.DCBA, 0));
	stProbe.fReal32_ABCD := LREAL_TO_REAL(F_MbDecode(pSrc, 2, E_MbType.Real32, E_MbWordOrder.ABCD, 0));
	stProbe.fReal32_CDAB := LREAL_TO_REAL(F_MbDecode(pSrc, 2, E_MbType.Real32, E_MbWordOrder.CDAB, 0));
	stProbe.fReal32_BADC := LREAL_TO_REAL(F_MbDecode(pSrc, 2, E_MbType.Real32, E_MbWordOrder.BADC, 0));
	stProbe.fReal32_DCBA := LREAL_TO_REAL(F_MbDecode(pSrc, 2, E_MbType.Real32, E_MbWordOrder.DCBA, 0));
END_IF
END_METHOD

METHOD PRIVATE FinishWrite
VAR_INPUT
	bOk    : BOOL;
	eClass : E_MbErrorClass;
	nExc   : BYTE;
END_VAR
VAR
	pPt    : POINTER TO ST_MbPoint;
END_VAR
pPt := aState[nCurWrite].pPoint;
IF pPt <> 0 THEN
	pPt^.bWriteBusy := FALSE;
	pPt^.bWriteDone := bOk;
	pPt^.bWriteErr  := NOT bOk;
END_IF
aState[nCurWrite].nWriteState := 3;
IF NOT bOk THEN
	WriteLog(nCurWrite, E_MbOp.Write, eClass, aState[nCurWrite].nWriteFc, nExc, nAttempt, 0);
END_IF
END_METHOD

METHOD PROTECTED Init
VAR
	i, j, nTmp : UINT;
	nKey       : UDINT;
	bOk        : BOOL;
END_VAR
bConfigError := FALSE;
bOk          := TRUE;
nBlocks      := 0;

IF eState <> E_MbDevState.Idle AND itfTransport <> 0 THEN
	itfTransport.Abort(nUnitId);
	itfTransport.Release(nUnitId);
END_IF
eState        := E_MbDevState.Idle;
nRotation     := 0;
nConsecFailTx := 0;
nDevRepeat    := 0;

IF bAddOverflow THEN
	ConfigFail(nPoints, GVL_MbConst.CFG_TOO_MANY_POINTS);
	bOk := FALSE;
END_IF
IF nPoints = 0 THEN
	ConfigFail(nPoints, GVL_MbConst.CFG_NO_POINTS);
	bInitDone := TRUE;
	RETURN;
END_IF

FOR i := 0 TO nPoints - 1 DO
	IF NOT ResolvePoint(i) THEN
		bOk := FALSE;
	END_IF
END_FOR

// Duplicate names and overlapping ranges. O(n²), runs once.
FOR i := 0 TO nPoints - 1 DO
	FOR j := i + 1 TO nPoints - 1 DO
		IF aState[i].sName = aState[j].sName THEN
			ConfigFail(j, GVL_MbConst.CFG_DUP_NAME);
			bOk := FALSE;
		END_IF
		IF aState[i].eRegion = aState[j].eRegion THEN
			IF UINT_TO_UDINT(aState[i].nOffset) < UINT_TO_UDINT(aState[j].nOffset) + aState[j].nCount
			   AND UINT_TO_UDINT(aState[j].nOffset) < UINT_TO_UDINT(aState[i].nOffset) + aState[i].nCount THEN
				ConfigFail(j, GVL_MbConst.CFG_OVERLAP);
				bOk := FALSE;
			END_IF
		END_IF
	END_FOR
END_FOR

IF bOk THEN
	// Insertion sort of point indices by SortKey
	FOR i := 0 TO nPoints - 1 DO
		aSorted[i] := i;
	END_FOR
	FOR i := 1 TO nPoints - 1 DO
		nTmp := aSorted[i];
		nKey := SortKey(nTmp);
		j    := i;
		WHILE j > 0 AND_THEN SortKey(aSorted[j - 1]) > nKey DO
			aSorted[j] := aSorted[j - 1];
			j := j - 1;
		END_WHILE
		aSorted[j] := nTmp;
	END_FOR

	IF NOT BuildBlocks() THEN
		bOk := FALSE;
	END_IF
END_IF

bConfigError := NOT bOk;
bInitDone    := TRUE;
END_METHOD

METHOD PRIVATE OnFailure
VAR_INPUT
	eClass     : E_MbErrorClass;
	nExc       : BYTE;
	bReachable : BOOL;    // TRUE when the device did answer (exception)
END_VAR
IF nAttempt < nRetries THEN
	nAttempt := nAttempt + 1;
	itfTransport.Abort(nUnitId);
	IF StartTx() THEN
		RETURN;
	END_IF
	eClass := E_MbErrorClass.Transport;
END_IF
IF bWriteTx THEN
	FinishWrite(FALSE, eClass, nExc);
ELSE
	FailBlock(eClass, nExc);
END_IF
EndTransaction(bReachable, eClass, nExc);
END_METHOD

METHOD PRIVATE OnResponse
nRxCount       := nRxCount + 1;
tLastRoundTrip := UDINT_TO_TIME(ULINT_TO_UDINT((tNow - tTxStart) / 10000));

IF bWriteTx THEN
	F_MbParseResponse(itfTransport.pResponsePdu, itfTransport.cbResponsePdu,
	                  aState[nCurWrite].nWriteFc, aState[nCurWrite].nWriteQty, stParse);
	IF stParse.bOk THEN
		FinishWrite(TRUE, E_MbErrorClass.None, 0);
		EndTransaction(TRUE, E_MbErrorClass.None, 0);
	ELSIF stParse.bException THEN
		IF stParse.nExcCode = 6 THEN
			OnFailure(E_MbErrorClass.Exception, 6, TRUE);
		ELSE
			FinishWrite(FALSE, E_MbErrorClass.Exception, stParse.nExcCode);
			EndTransaction(TRUE, E_MbErrorClass.None, 0);
		END_IF
	ELSE
		OnFailure(stParse.eClass, 0, FALSE);
	END_IF
	RETURN;
END_IF

F_MbParseResponse(itfTransport.pResponsePdu, itfTransport.cbResponsePdu,
                  aBlocks[nCurBlock].nFc, aBlocks[nCurBlock].nCount, stParse);

IF stParse.bOk THEN
	ScatterBlock();
	EndTransaction(TRUE, E_MbErrorClass.None, 0);
ELSIF stParse.bException THEN
	// The device answered, so it is reachable whatever it said
	IF (stParse.nExcCode = 2 OR stParse.nExcCode = 3) AND_THEN SplitBlock(nCurBlock) THEN
		WriteLog(aSorted[aBlocks[nCurBlock].nSortedFirst], E_MbOp.Read, E_MbErrorClass.Exception,
		         aBlocks[nCurBlock].nFc, stParse.nExcCode, nAttempt, 0);
		EndTransaction(TRUE, E_MbErrorClass.None, 0);
	ELSIF stParse.nExcCode = 6 THEN
		OnFailure(E_MbErrorClass.Exception, 6, TRUE);        // Busy: worth a retry
	ELSE
		FailBlock(E_MbErrorClass.Exception, stParse.nExcCode);
		EndTransaction(TRUE, E_MbErrorClass.None, 0);
	END_IF
ELSE
	OnFailure(stParse.eClass, 0, FALSE);                       // Truncated / Malformed
END_IF
END_METHOD

METHOD PUBLIC Profile
VAR_INPUT
	sModel          : STRING;
	eWordOrder      : E_MbWordOrder  := E_MbWordOrder.ABCD;
	eAddressing     : E_MbAddressing := E_MbAddressing.Modicon;
	nMaxRegsPerRead : UINT := 125;
	nMaxGap         : UINT := 8;
	bFc6Only        : BOOL := FALSE;
	bFc16Only       : BOOL := FALSE;
	bStringByteSwap : BOOL := FALSE;
	tSlowPoll       : TIME := T#5S;
END_VAR
VAR
	sModelTrunc : STRING(GVL_MbParam.MB_NAME_LEN);
END_VAR
// Called every cycle from the profile's body. Only a real change triggers re-initialization.
sModelTrunc := sModel;
IF stProfile.sModel <> sModelTrunc OR stProfile.eWordOrder <> eWordOrder OR stProfile.eAddressing <> eAddressing
   OR stProfile.nMaxRegsPerRead <> LIMIT(1, nMaxRegsPerRead, GVL_MbConst.MAX_READ_REGS)
   OR stProfile.nMaxGap <> nMaxGap OR stProfile.bFc6Only <> bFc6Only OR stProfile.bFc16Only <> bFc16Only
   OR stProfile.bStringByteSwap <> bStringByteSwap OR stProfile.tSlowPoll <> tSlowPoll THEN
	stProfile.sModel          := sModelTrunc;
	stProfile.eWordOrder      := eWordOrder;
	stProfile.eAddressing     := eAddressing;
	stProfile.nMaxRegsPerRead := LIMIT(1, nMaxRegsPerRead, GVL_MbConst.MAX_READ_REGS);
	stProfile.nMaxGap         := nMaxGap;
	stProfile.bFc6Only        := bFc6Only;
	stProfile.bFc16Only       := bFc16Only;
	stProfile.bStringByteSwap := bStringByteSwap;
	stProfile.tSlowPoll       := tSlowPoll;
	bRegChanged := TRUE;
END_IF
nRegCursor   := 0;
bAddOverflow := FALSE;
END_METHOD

METHOD PRIVATE RecomputeBlockRange
VAR_INPUT
	nB : UINT;
END_VAR
VAR
	k, nFirst, nLast : UINT;
END_VAR
// Points are sorted and non-overlapping, so the last point's end is the block end
nFirst := aSorted[aBlocks[nB].nSortedFirst];
nLast  := aSorted[aBlocks[nB].nSortedFirst + aBlocks[nB].nSortedCount - 1];
aBlocks[nB].nOffset     := aState[nFirst].nOffset;
aBlocks[nB].nCount      := aState[nLast].nOffset + aState[nLast].nCount - aState[nFirst].nOffset;
aBlocks[nB].nConsecFail := 0;
aBlocks[nB].tLastPoll   := 0;
FOR k := 0 TO aBlocks[nB].nSortedCount - 1 DO
	aState[aSorted[aBlocks[nB].nSortedFirst + k]].nBlock := nB;
END_FOR
END_METHOD

METHOD PROTECTED ResolvePoint : BOOL
VAR_INPUT
	i     : UINT;
END_VAR
VAR
	pP    	: POINTER TO ST_MbPoint;
	eReg  	: E_MbRegion;
	nOff  	: UDINT;
	bBits 	: BOOL;
	bOk   	: BOOL;
	bRange	: BOOL;
	bGain 	: BOOL;
END_VAR
ResolvePoint := FALSE;
bOk := TRUE;
pP  := aState[i].pPoint;

IF pP = 0 OR_ELSE pP^.wMagic <> 16#4D50 THEN
	ConfigFail(i, GVL_MbConst.CFG_BAD_MAGIC);
	RETURN;
END_IF
IF LEN(aState[i].sName) = 0 THEN
	ConfigFail(i, GVL_MbConst.CFG_EMPTY_NAME);
	bOk := FALSE;
END_IF

// ---- Region and 0-based offset ----
eReg := E_MbRegion.Auto;
nOff := 0;
CASE stProfile.eAddressing OF
	E_MbAddressing.Modicon:
		IF pP^.nAddr >= 1 AND pP^.nAddr <= 9999 THEN
			eReg := E_MbRegion.Coil;            nOff := pP^.nAddr - 1;
		ELSIF pP^.nAddr >= 10001 AND pP^.nAddr <= 19999 THEN
			eReg := E_MbRegion.DiscreteInput;   nOff := pP^.nAddr - 10001;
		ELSIF pP^.nAddr >= 30001 AND pP^.nAddr <= 39999 THEN
			eReg := E_MbRegion.InputRegister;   nOff := pP^.nAddr - 30001;
		ELSIF pP^.nAddr >= 40001 AND pP^.nAddr <= 49999 THEN
			eReg := E_MbRegion.HoldingRegister; nOff := pP^.nAddr - 40001;
		ELSIF pP^.nAddr >= 100001 AND pP^.nAddr <= 165536 THEN
			eReg := E_MbRegion.DiscreteInput;   nOff := pP^.nAddr - 100001;
		ELSIF pP^.nAddr >= 300001 AND pP^.nAddr <= 365536 THEN
			eReg := E_MbRegion.InputRegister;   nOff := pP^.nAddr - 300001;
		ELSIF pP^.nAddr >= 400001 AND pP^.nAddr <= 465536 THEN
			eReg := E_MbRegion.HoldingRegister; nOff := pP^.nAddr - 400001;
		END_IF
		IF eReg = E_MbRegion.Auto THEN
			ConfigFail(i, GVL_MbConst.CFG_BAD_ADDRESS);
			bOk := FALSE;
		ELSIF pP^.eRegion <> E_MbRegion.Auto AND pP^.eRegion <> eReg THEN
			ConfigFail(i, GVL_MbConst.CFG_REGION_MISMATCH);
			bOk := FALSE;
		END_IF

	E_MbAddressing.Offset0:
		eReg := pP^.eRegion;
		nOff := pP^.nAddr;

	E_MbAddressing.Offset1:
		eReg := pP^.eRegion;
		IF pP^.nAddr >= 1 THEN
			nOff := pP^.nAddr - 1;
		ELSE
			ConfigFail(i, GVL_MbConst.CFG_BAD_ADDRESS);
			bOk := FALSE;
		END_IF
END_CASE

IF eReg = E_MbRegion.Auto THEN
	IF stProfile.eAddressing <> E_MbAddressing.Modicon THEN
		ConfigFail(i, GVL_MbConst.CFG_REGION_REQUIRED);
	END_IF
	bOk  := FALSE;
	eReg := E_MbRegion.HoldingRegister;   // Keep the remaining checks meaningful
END_IF
IF nOff > 65535 THEN
	ConfigFail(i, GVL_MbConst.CFG_BAD_ADDRESS);
	bOk  := FALSE;
	nOff := 0;
END_IF
bBits := (eReg = E_MbRegion.Coil) OR (eReg = E_MbRegion.DiscreteInput);

// ---- Type and register count ----
aState[i].eType := pP^.eType;
IF aState[i].eType = E_MbType.Auto THEN
	IF bBits THEN
		aState[i].eType := E_MbType.Boolean;
	ELSE
		aState[i].eType := E_MbType.UInt16;
	END_IF
END_IF
aState[i].nCount := 1;
CASE aState[i].eType OF
	E_MbType.Boolean:
		IF NOT bBits THEN
			ConfigFail(i, GVL_MbConst.CFG_BAD_TYPE);
			bOk := FALSE;
		END_IF
	E_MbType.Int16, E_MbType.UInt16:
		IF bBits THEN
			ConfigFail(i, GVL_MbConst.CFG_BAD_TYPE);
			bOk := FALSE;
		END_IF
	E_MbType.RegisterBit:
		IF bBits THEN
			ConfigFail(i, GVL_MbConst.CFG_BAD_TYPE);
			bOk := FALSE;
		END_IF
		IF pP^.nBit > 15 THEN
			ConfigFail(i, GVL_MbConst.CFG_BAD_BIT);
			bOk := FALSE;
		END_IF
	E_MbType.Int32, E_MbType.UInt32, E_MbType.Real32:
		IF bBits THEN
			ConfigFail(i, GVL_MbConst.CFG_BAD_TYPE);
			bOk := FALSE;
		END_IF
		aState[i].nCount := 2;
	E_MbType.Int64, E_MbType.UInt64, E_MbType.Real64:
		IF bBits THEN
			ConfigFail(i, GVL_MbConst.CFG_BAD_TYPE);
			bOk := FALSE;
		END_IF
		aState[i].nCount := 4;
	E_MbType.Text:
		IF bBits OR pP^.nRegs < 1 OR pP^.nRegs > GVL_MbParam.MB_STR_LEN / 2 THEN
			ConfigFail(i, GVL_MbConst.CFG_BAD_REGS);
			bOk := FALSE;
		ELSE
			aState[i].nCount := pP^.nRegs;
		END_IF
	E_MbType.Raw:
		IF bBits OR pP^.nRegs < 1 OR pP^.nRegs > GVL_MbParam.MB_RAW_WORDS THEN
			ConfigFail(i, GVL_MbConst.CFG_BAD_REGS);
			bOk := FALSE;
		ELSE
			aState[i].nCount := pP^.nRegs;
		END_IF
END_CASE
IF NOT bBits AND aState[i].nCount > stProfile.nMaxRegsPerRead THEN
	ConfigFail(i, GVL_MbConst.CFG_BAD_REGS);
	bOk := FALSE;
END_IF
IF nOff + aState[i].nCount > 65536 THEN
	ConfigFail(i, GVL_MbConst.CFG_BAD_ADDRESS);
	bOk := FALSE;
END_IF

// ---- Scaling and fail value ----
bRange := pP^.fRawMin <> pP^.fRawMax;
bGain  := pP^.fGain <> 0 OR pP^.fOffset <> 0;
IF bRange AND bGain THEN
	ConfigFail(i, GVL_MbConst.CFG_BAD_SCALING);   // One form or the other
	bOk := FALSE;
END_IF
IF bGain AND pP^.fGain = 0 THEN
	ConfigFail(i, GVL_MbConst.CFG_BAD_SCALING);   // Offset without gain; use fGain := 1 for offset only
	bOk := FALSE;
END_IF
IF bRange AND pP^.fEngMin = pP^.fEngMax THEN
	ConfigFail(i, GVL_MbConst.CFG_BAD_SCALING);
	bOk := FALSE;
END_IF
IF NOT bRange AND (pP^.fEngMin <> 0 OR pP^.fEngMax <> 0) THEN
	ConfigFail(i, GVL_MbConst.CFG_BAD_SCALING);   // Eng range given without a raw range
	bOk := FALSE;
END_IF
IF (bRange OR bGain) AND (aState[i].eType = E_MbType.Boolean OR aState[i].eType = E_MbType.RegisterBit
   OR aState[i].eType = E_MbType.Text OR aState[i].eType = E_MbType.Raw) THEN
	ConfigFail(i, GVL_MbConst.CFG_BAD_SCALING);
	bOk := FALSE;
END_IF
IF pP^.bUseFailValue AND (aState[i].eType = E_MbType.Text OR aState[i].eType = E_MbType.Raw) THEN
	ConfigFail(i, GVL_MbConst.CFG_BAD_FAILVALUE);
	bOk := FALSE;
END_IF

// ---- Word order ----
aState[i].eWordOrder := pP^.eWordOrder;
IF aState[i].eWordOrder = E_MbWordOrder.Inherit THEN
	aState[i].eWordOrder := stProfile.eWordOrder;
END_IF
IF aState[i].eWordOrder = E_MbWordOrder.Inherit THEN
	aState[i].eWordOrder := E_MbWordOrder.ABCD;
END_IF

// ---- Function codes ----
aState[i].nWriteFc := 0;
CASE eReg OF
	E_MbRegion.Coil:
		aState[i].nReadFc  := GVL_MbConst.FC_READ_COILS;
		aState[i].nWriteFc := SEL(stProfile.bFc16Only, GVL_MbConst.FC_WRITE_COIL, GVL_MbConst.FC_WRITE_COILS);
	E_MbRegion.DiscreteInput:
		aState[i].nReadFc  := GVL_MbConst.FC_READ_DISCRETE;
	E_MbRegion.InputRegister:
		aState[i].nReadFc  := GVL_MbConst.FC_READ_INPUT;
	E_MbRegion.HoldingRegister:
		aState[i].nReadFc  := GVL_MbConst.FC_READ_HOLDING;
		IF aState[i].nCount = 1 THEN
			aState[i].nWriteFc := SEL(stProfile.bFc16Only, GVL_MbConst.FC_WRITE_REGISTER, GVL_MbConst.FC_WRITE_REGISTERS);
		ELSIF NOT stProfile.bFc6Only THEN
			aState[i].nWriteFc := GVL_MbConst.FC_WRITE_REGISTERS;
		END_IF
END_CASE
// Text/Raw are read-only in v1; a bit write would need read-modify-write, also not in v1
IF aState[i].eType = E_MbType.Text OR aState[i].eType = E_MbType.Raw OR aState[i].eType = E_MbType.RegisterBit THEN
	aState[i].nWriteFc := 0;
END_IF

// ---- Store, reset runtime state ----
aState[i].eRegion     := eReg;
aState[i].nOffset     := UDINT_TO_UINT(nOff);
aState[i].nBlock      := GVL_MbParam.MB_MAX_BLOCKS;
aState[i].bFailing    := FALSE;
aState[i].nRepeat     := 0;
aState[i].tLastLog    := 0;
aState[i].eLastClass  := E_MbErrorClass.None;
aState[i].nLastExc    := 0;
aState[i].nWriteState := 0;

IF NOT bOk THEN
	aState[i].nCount := 0;   // Failed points occupy no range; keeps them out of the overlap check
END_IF
ResolvePoint := bOk;
END_METHOD

METHOD PRIVATE ScatterBlock
VAR
	k, idx, nRel : UINT;
	pData        : POINTER TO BYTE;
	pPt          : POINTER TO ST_MbPoint;
	bBits        : BOOL;
END_VAR
pData := itfTransport.pResponsePdu + stParse.nDataOffset;
bBits := (aBlocks[nCurBlock].eRegion = E_MbRegion.Coil) OR (aBlocks[nCurBlock].eRegion = E_MbRegion.DiscreteInput);

FOR k := 0 TO aBlocks[nCurBlock].nSortedCount - 1 DO
	idx := aSorted[aBlocks[nCurBlock].nSortedFirst + k];
	pPt := aState[idx].pPoint;
	IF pPt = 0 THEN
		CONTINUE;
	END_IF
	nRel := aState[idx].nOffset - aBlocks[nCurBlock].nOffset;
	IF bBits THEN
		pPt^.fValue  := SEL((pData[nRel / 8] AND SHL(BYTE#1, nRel MOD 8)) <> 0, 0.0, 1.0);
		pPt^.aRaw[0] := SEL(pPt^.fValue <> 0, WORD#0, WORD#1);
	ELSE
		DecodePoint(idx, pData + 2 * nRel);
	END_IF
	pPt^.bValid    := TRUE;
	pPt^.tLastGood := tNow;
END_FOR

// Block recovered? The first point carries the block's flood-control state.
idx := aSorted[aBlocks[nCurBlock].nSortedFirst];
IF aState[idx].bFailing THEN
	aState[idx].bFailing := FALSE;
	IF bOnline THEN
		WriteLog(idx, E_MbOp.Read, E_MbErrorClass.Recovered, aBlocks[nCurBlock].nFc, 0, 0, aState[idx].nRepeat);
	END_IF
	aState[idx].nRepeat := 0;
END_IF
aBlocks[nCurBlock].nConsecFail := 0;
aBlocks[nCurBlock].tLastPoll   := tNow;
END_METHOD

METHOD PRIVATE Scheduler
VAR
	eXfer : E_MbXferState;
END_VAR
IF eState = E_MbDevState.Cooldown THEN
	eState := E_MbDevState.Idle;          // One-cycle gap after Release keeps arbitration fair
	RETURN;
END_IF

IF eState = E_MbDevState.Idle THEN
	IF SelectNextWrite() THEN
		bWriteTx := TRUE;                     // Writes preempt the read rotation and ignore backoff
	ELSE
		IF NOT bOnline AND tNow < tNextPoll THEN
			RETURN;
		END_IF
		IF NOT SelectNextBlock() THEN
			RETURN;
		END_IF
		bWriteTx := FALSE;
	END_IF
	eState := E_MbDevState.Acquire;
END_IF

IF eState = E_MbDevState.Acquire THEN
	IF NOT itfTransport.Acquire(nUnitId) THEN
		RETURN;
	END_IF
	nAttempt := 0;
	IF NOT StartTx() THEN
		IF bWriteTx THEN
			FinishWrite(FALSE, E_MbErrorClass.Transport, 0);
		END_IF
		EndTransaction(FALSE, E_MbErrorClass.Transport, 0);
	END_IF
	RETURN;
END_IF

IF eState = E_MbDevState.Wait THEN
	eXfer := itfTransport.Poll();
	CASE eXfer OF
		E_MbXferState.Done:    OnResponse();
		E_MbXferState.Timeout: OnFailure(E_MbErrorClass.Timeout, 0, FALSE);
		E_MbXferState.Error:   OnFailure(itfTransport.eLastError, 0, FALSE);
		E_MbXferState.Idle:    OnFailure(E_MbErrorClass.Transport, 0, FALSE);
	END_CASE
END_IF
END_METHOD

METHOD PRIVATE SelectNextBlock : BOOL
VAR
	k, nB : UINT;
	tSlow : ULINT;
END_VAR
SelectNextBlock := FALSE;
IF nBlocks = 0 THEN
	RETURN;
END_IF
tSlow := F_MbTimeToFt(stProfile.tSlowPoll);
FOR k := 0 TO nBlocks - 1 DO
	nB := (nRotation + k) MOD nBlocks;
	IF aBlocks[nB].ePoll = E_MbPoll.Fast OR_ELSE (tNow - aBlocks[nB].tLastPoll >= tSlow) THEN
		nCurBlock       := nB;
		nRotation       := (nB + 1) MOD nBlocks;
		SelectNextBlock := TRUE;
		RETURN;
	END_IF
END_FOR
END_METHOD

METHOD PRIVATE SelectNextWrite : BOOL
VAR
	i : UINT;
END_VAR
SelectNextWrite := FALSE;
FOR i := 0 TO nPoints - 1 DO
	IF aState[i].nWriteState = 1 THEN
		nCurWrite             := i;
		aState[i].nWriteState := 2;
		SelectNextWrite       := TRUE;
		RETURN;
	END_IF
END_FOR
END_METHOD

METHOD PRIVATE ServiceWrites
VAR
	i   : UINT;
	pPt : POINTER TO ST_MbPoint;
END_VAR
// Handshake: bWriteReq rises -> queued (Busy) -> Done or Err held until bWriteReq drops
IF nPoints = 0 THEN
	RETURN;
END_IF
FOR i := 0 TO nPoints - 1 DO
	pPt := aState[i].pPoint;
	IF pPt = 0 THEN
		CONTINUE;
	END_IF
	CASE aState[i].nWriteState OF
		0:
			IF pPt^.bWriteReq THEN
				pPt^.bWriteDone := FALSE;
				pPt^.bWriteErr  := FALSE;
				IF aState[i].nWriteFc = 0 THEN
					pPt^.bWriteErr        := TRUE;
					aState[i].nWriteState := 3;
					WriteLog(i, E_MbOp.Write, E_MbErrorClass.Config, 0, GVL_MbConst.CFG_NOT_WRITABLE, 0, 0);
				ELSIF NOT EncodeWrite(i) THEN
					pPt^.bWriteErr        := TRUE;
					aState[i].nWriteState := 3;
					WriteLog(i, E_MbOp.Write, E_MbErrorClass.Config, aState[i].nWriteFc, GVL_MbConst.CFG_WRITE_RANGE, 0, 0);
				ELSE
					pPt^.bWriteBusy       := TRUE;
					aState[i].nWriteState := 1;
				END_IF
			END_IF
		3:
			IF NOT pPt^.bWriteReq THEN
				pPt^.bWriteDone       := FALSE;
				pPt^.bWriteErr        := FALSE;
				pPt^.bWriteBusy       := FALSE;
				aState[i].nWriteState := 0;
			END_IF
	END_CASE
END_FOR
END_METHOD

METHOD PROTECTED SortKey : UDINT
VAR_INPUT
	i    : UINT;
END_VAR
VAR
	nKey : UDINT;
END_VAR
// (poll class, region, offset) packed so an integer compare yields block-building order
nKey := 0;
IF aState[i].pPoint <> 0 THEN
	CASE aState[i].pPoint^.ePoll OF
		E_MbPoll.Fast: nKey := 0;
		E_MbPoll.Slow: nKey := 1;
		E_MbPoll.Off:  nKey := 2;
	END_CASE
END_IF
nKey := nKey * 4;
CASE aState[i].eRegion OF
	E_MbRegion.Coil:            nKey := nKey + 0;
	E_MbRegion.DiscreteInput:   nKey := nKey + 1;
	E_MbRegion.InputRegister:   nKey := nKey + 2;
	E_MbRegion.HoldingRegister: nKey := nKey + 3;
END_CASE
SortKey := SHL(nKey, 16) + aState[i].nOffset;
END_METHOD

METHOD PRIVATE SplitBlock : BOOL
VAR_INPUT
	nB    : UINT;
END_VAR
VAR
	n     : INT;
	k     : UINT;
	nHalf : UINT;
END_VAR
SplitBlock := FALSE;
IF nB >= nBlocks OR aBlocks[nB].nSortedCount < 2 OR nBlocks >= GVL_MbParam.MB_MAX_BLOCKS THEN
	RETURN;   // A single multi-register point can't be split; it just keeps failing
END_IF

// Make room at nB+1
FOR n := UINT_TO_INT(nBlocks) TO UINT_TO_INT(nB) + 2 BY -1 DO
	aBlocks[n] := aBlocks[n - 1];
END_FOR
nBlocks := nBlocks + 1;
FOR k := 0 TO nPoints - 1 DO
	IF aState[k].nBlock > nB AND aState[k].nBlock < GVL_MbParam.MB_MAX_BLOCKS THEN
		aState[k].nBlock := aState[k].nBlock + 1;
	END_IF
END_FOR

// Halve the point range; recompute both address ranges
nHalf := aBlocks[nB].nSortedCount / 2;
aBlocks[nB + 1]              := aBlocks[nB];
aBlocks[nB + 1].nSortedFirst := aBlocks[nB].nSortedFirst + nHalf;
aBlocks[nB + 1].nSortedCount := aBlocks[nB].nSortedCount - nHalf;
aBlocks[nB].nSortedCount     := nHalf;
RecomputeBlockRange(nB);
RecomputeBlockRange(nB + 1);
SplitBlock := TRUE;
END_METHOD

METHOD PRIVATE StartRead : BOOL
StartRead := FALSE;
cbPdu := F_MbBuildRequest(aBlocks[nCurBlock].nFc, aBlocks[nCurBlock].nOffset, aBlocks[nCurBlock].nCount,
                          0, 0, ADR(aPdu), GVL_MbParam.MB_ADU_SIZE);
IF cbPdu = 0 THEN
	RETURN;
END_IF
nExpectedLen := F_MbExpectedResponseLength(aBlocks[nCurBlock].nFc, aBlocks[nCurBlock].nCount);
IF NOT itfTransport.Send(nUnitId, ADR(aPdu), cbPdu, nExpectedLen, tTimeout) THEN
	RETURN;
END_IF
tTxStart  := tNow;
nTxCount  := nTxCount + 1;
eState    := E_MbDevState.Wait;
StartRead := TRUE;
END_METHOD

METHOD PRIVATE StartTx : BOOL
IF bWriteTx THEN
	StartTx := StartWrite();
ELSE
	StartTx := StartRead();
END_IF
END_METHOD

METHOD PRIVATE StartWrite : BOOL
StartWrite := FALSE;
cbPdu := F_MbBuildRequest(aState[nCurWrite].nWriteFc, aState[nCurWrite].nOffset, aState[nCurWrite].nWriteQty,
                          ADR(aState[nCurWrite].aWriteData), aState[nCurWrite].cbWriteData,
                          ADR(aPdu), GVL_MbParam.MB_ADU_SIZE);
IF cbPdu = 0 THEN
	RETURN;
END_IF
nExpectedLen := F_MbExpectedResponseLength(aState[nCurWrite].nWriteFc, aState[nCurWrite].nWriteQty);
IF NOT itfTransport.Send(nUnitId, ADR(aPdu), cbPdu, nExpectedLen, tTimeout) THEN
	RETURN;
END_IF
tTxStart   := tNow;
nTxCount   := nTxCount + 1;
eState     := E_MbDevState.Wait;
StartWrite := TRUE;
END_METHOD

METHOD PROTECTED WriteLog
VAR_INPUT
	nPointIdx : UINT;              // >= nPoints means device-level entry
	eOp       : E_MbOp;
	eClass    : E_MbErrorClass;
	nFc       : USINT;
	nExcCode  : BYTE;
	nRetries  : USINT;
	nRepeat   : UDINT;
END_VAR
VAR
	stEntry   : ST_MbLogEntry;
END_VAR
IF pLog = 0 THEN
	nLogDropped := nLogDropped + 1;
	RETURN;
END_IF

stEntry.tTime    := tNow;
stEntry.nUnitId  := nUnitId;
stEntry.eOp      := eOp;
stEntry.eClass   := eClass;
stEntry.nFc      := USINT_TO_BYTE(nFc);
stEntry.nExcCode := nExcCode;
stEntry.nRetries := nRetries;
stEntry.nRepeat  := nRepeat;

IF nPointIdx < nPoints AND aState[nPointIdx].pPoint <> 0 THEN
	stEntry.sName   := aState[nPointIdx].sName;
	stEntry.eRegion := aState[nPointIdx].eRegion;
	stEntry.nAddr   := aState[nPointIdx].pPoint^.nAddr;
ELSE
	stEntry.sName   := stProfile.sModel;
END_IF

// Ring insert
IF pLog^.nHead >= GVL_MbParam.MB_LOG_SIZE THEN
	pLog^.nHead := 0;
END_IF
pLog^.aEntries[pLog^.nHead] := stEntry;
pLog^.nHead := (pLog^.nHead + 1) MOD GVL_MbParam.MB_LOG_SIZE;
IF pLog^.nCount < GVL_MbParam.MB_LOG_SIZE THEN
	pLog^.nCount := pLog^.nCount + 1;
ELSE
	pLog^.nDropped := pLog^.nDropped + 1;
END_IF
pLog^.nSeq := pLog^.nSeq + 1;

IF eClass <> E_MbErrorClass.Recovered AND eClass <> E_MbErrorClass.None THEN
	pLog^.nTotalErrors := pLog^.nTotalErrors + 1;
	nErrorCount        := nErrorCount + 1;
	stLastError        := stEntry;
END_IF
END_METHOD

END_FUNCTION_BLOCK

// ---- POUs/Log/FB_MbLogWriter.TcPOU
FUNCTION_BLOCK FB_MbLogWriter
VAR_INPUT
	bEnable   : BOOL := TRUE;
	sDir      : STRING(255);              // Folder; trailing backslash optional; created if missing
	sName     : STRING(80);               // File name without extension
	pLog      : POINTER TO ST_MbLog;      // Ring to drain; the owner refreshes this every cycle
	tNow      : ULINT;                    // FILETIME from the owner
END_VAR
VAR_OUTPUT
	bError    : BOOL;                     // File trouble; retried every MB_LOG_FILE_RETRY
	nErrId    : UDINT;
	nWritten  : UDINT;                    // Entries appended since start
	nDropped  : UDINT;                    // Entries that scrolled out of the ring unwritten
	sFile     : STRING(255);
END_VAR
VAR
	eStep        : E_MbLogWriterStep;
	fbMkDir      : FB_CreateDir;
	fbOpen       : FB_FileOpen;
	fbSeek       : FB_FileSeek;
	fbTell       : FB_FileTell;
	fbPuts       : FB_FilePuts;
	fbClose      : FB_FileClose;
	fbDelete     : FB_FileDelete;
	fbRename     : FB_FileRename;
	hFile        : UINT;
	bStarted     : BOOL;
	nCursor      : UDINT;                 // Next sequence number to write
	nPending     : UDINT;
	nInBatch     : USINT;
	nSize        : UDINT;
	bDirDone     : BOOL;
	nDirPos      : INT;
	sDirNorm     : STRING(255);
	sDirPrev     : STRING(255);
	sFileOld     : STRING(255);
	sLine        : STRING(255);
	bLineIsEntry : BOOL;
	bRotate      : BOOL;
	bFailClose   : BOOL;
	tRetryAt     : ULINT;
	pDir         : POINTER TO BYTE;
	i            : INT;
END_VAR

IF NOT bEnable OR pLog = 0 THEN
	RETURN;
END_IF
IF NOT bStarted THEN
	bStarted := TRUE;
	nCursor  := pLog^.nSeq;                  // Don't replay what was in the ring before we started
END_IF

// Pending entries; if the ring outran us, skip to what is still there and count the loss
nPending := pLog^.nSeq - nCursor;
IF nPending > GVL_MbParam.MB_LOG_SIZE THEN
	nDropped := nDropped + (nPending - GVL_MbParam.MB_LOG_SIZE);
	nCursor  := pLog^.nSeq - GVL_MbParam.MB_LOG_SIZE;
	nPending := GVL_MbParam.MB_LOG_SIZE;
END_IF

CASE eStep OF
	E_MbLogWriterStep.Idle:
		IF nPending = 0 OR tNow < tRetryAt THEN
			RETURN;
		END_IF
		BuildNames();
		IF NOT bDirDone THEN
			nDirPos := 3;                        // Skip the drive letter and its backslash
			eStep   := E_MbLogWriterStep.MkDir;
		ELSE
			eStep := E_MbLogWriterStep.Open;
		END_IF

	E_MbLogWriterStep.MkDir:
		// Create the next path prefix (each level separately)
		pDir := ADR(sDirNorm);
		i := nDirPos;
		WHILE i < LEN(sDirNorm) AND_THEN pDir[i] <> 16#5C DO      // '\'
			i := i + 1;
		END_WHILE
		IF i >= LEN(sDirNorm) THEN
			bDirDone := TRUE;
			eStep    := E_MbLogWriterStep.Open;
		ELSE
			fbMkDir(sNetId := '', sPathName := LEFT(sDirNorm, i), ePath := PATH_GENERIC, bExecute := TRUE, tTimeout := T#5S);
			nDirPos := i + 1;
			eStep   := E_MbLogWriterStep.MkDirWait;
		END_IF

	E_MbLogWriterStep.MkDirWait:
		fbMkDir(bExecute := FALSE);
		IF NOT fbMkDir.bBusy THEN
			eStep := E_MbLogWriterStep.MkDir;    // Errors ignored: "exists" is fine, anything real surfaces at Open
		END_IF

	E_MbLogWriterStep.Open:
		fbOpen(sNetId := '', sPathName := sFile, nMode := FOPEN_MODEAPPEND OR FOPEN_MODETEXT,
		       ePath := PATH_GENERIC, bExecute := TRUE, tTimeout := T#5S);
		eStep := E_MbLogWriterStep.OpenWait;

	E_MbLogWriterStep.OpenWait:
		fbOpen(bExecute := FALSE);
		IF NOT fbOpen.bBusy THEN
			IF fbOpen.bError THEN
				Fail(fbOpen.nErrId, FALSE);
			ELSE
				hFile := fbOpen.hFile;
				fbSeek(sNetId := '', hFile := hFile, nSeekPos := 0, eOrigin := SEEK_END, bExecute := TRUE, tTimeout := T#5S);
				eStep := E_MbLogWriterStep.SeekWait;
			END_IF
		END_IF

	E_MbLogWriterStep.SeekWait:
		fbSeek(bExecute := FALSE);
		IF NOT fbSeek.bBusy THEN
			IF fbSeek.bError THEN
				Fail(fbSeek.nErrId, TRUE);
			ELSE
				fbTell(sNetId := '', hFile := hFile, bExecute := TRUE, tTimeout := T#5S);
				eStep := E_MbLogWriterStep.TellWait;
			END_IF
		END_IF

	E_MbLogWriterStep.TellWait:
		fbTell(bExecute := FALSE);
		IF NOT fbTell.bBusy THEN
			IF fbTell.bError THEN
				Fail(fbTell.nErrId, TRUE);
			ELSE
				nSize    := DINT_TO_UDINT(MAX(0, fbTell.nSeekPos));
				nInBatch := 0;
				IF nSize >= GVL_MbParam.MB_LOG_FILE_MAX_BYTES THEN
					bRotate := TRUE;
					fbClose(sNetId := '', hFile := hFile, bExecute := TRUE, tTimeout := T#5S);
					eStep := E_MbLogWriterStep.CloseWait;
				ELSE
					IF nSize = 0 THEN
						sLine := 'TimeUTC,Name,Unit,Region,Address,FC,Op,Class,ExcCode,Retries,Repeat$N';
						bLineIsEntry := FALSE;
					ELSE
						sLine := NextLine();
					END_IF
					fbPuts(sNetId := '', hFile := hFile, sLine := sLine, bExecute := TRUE, tTimeout := T#5S);
					eStep := E_MbLogWriterStep.PutWait;
				END_IF
			END_IF
		END_IF

	E_MbLogWriterStep.PutWait:
		fbPuts(bExecute := FALSE);
		IF NOT fbPuts.bBusy THEN
			IF fbPuts.bError THEN
				Fail(fbPuts.nErrId, TRUE);
			ELSE
				nSize := nSize + INT_TO_UDINT(LEN(sLine)) + 1;           // +1: the LF becomes CRLF in text mode
				IF bLineIsEntry THEN
					nCursor  := nCursor + 1;
					nWritten := nWritten + 1;
					nInBatch := nInBatch + 1;
				END_IF
				nPending := pLog^.nSeq - nCursor;
				IF nPending > 0 AND nInBatch < GVL_MbParam.MB_LOG_FILE_BATCH AND nSize < GVL_MbParam.MB_LOG_FILE_MAX_BYTES THEN
					sLine := NextLine();
					fbPuts(sNetId := '', hFile := hFile, sLine := sLine, bExecute := TRUE, tTimeout := T#5S);
				ELSE
					fbClose(sNetId := '', hFile := hFile, bExecute := TRUE, tTimeout := T#5S);
					eStep := E_MbLogWriterStep.CloseWait;
				END_IF
			END_IF
		END_IF

	E_MbLogWriterStep.CloseWait:
		fbClose(bExecute := FALSE);
		IF NOT fbClose.bBusy THEN
			hFile := 0;
			IF bFailClose THEN
				bFailClose := FALSE;
				eStep := E_MbLogWriterStep.Idle;                          // tRetryAt was set by Fail
			ELSIF bRotate THEN
				fbDelete(sNetId := '', sPathName := sFileOld, ePath := PATH_GENERIC, bExecute := TRUE, tTimeout := T#5S);
				eStep := E_MbLogWriterStep.DeleteWait;
			ELSE
				bError := FALSE;
				eStep  := E_MbLogWriterStep.Idle;
			END_IF
		END_IF

	E_MbLogWriterStep.DeleteWait:
		fbDelete(bExecute := FALSE);
		IF NOT fbDelete.bBusy THEN                                        // "not found" is fine
			fbRename(sNetId := '', sOldName := sFile, sNewName := sFileOld, ePath := PATH_GENERIC, bExecute := TRUE, tTimeout := T#5S);
			eStep := E_MbLogWriterStep.RenameWait;
		END_IF

	E_MbLogWriterStep.RenameWait:
		fbRename(bExecute := FALSE);
		IF NOT fbRename.bBusy THEN
			bRotate := FALSE;
			IF fbRename.bError THEN
				Fail(fbRename.nErrId, FALSE);
			ELSE
				eStep := E_MbLogWriterStep.Idle;                          // Next batch opens a fresh file with a header
			END_IF
		END_IF
END_CASE

METHOD PRIVATE BuildNames
sDirNorm := sDir;
IF LEN(sDirNorm) > 0 AND_THEN RIGHT(sDirNorm, 1) <> '\' THEN
	sDirNorm := CONCAT(sDirNorm, '\');
END_IF
IF sDirNorm <> sDirPrev THEN
	sDirPrev := sDirNorm;
	bDirDone := FALSE;
END_IF
sFile    := CONCAT(CONCAT(sDirNorm, sName), '.csv');
sFileOld := CONCAT(CONCAT(sDirNorm, sName), '.1.csv');
END_METHOD

METHOD PRIVATE Fail
VAR_INPUT
	nId         : UDINT;
	bCloseFirst : BOOL;
END_VAR
bError   := TRUE;
nErrId   := nId;
tRetryAt := tNow + F_MbTimeToFt(GVL_MbParam.MB_LOG_FILE_RETRY);
bRotate  := FALSE;
IF bCloseFirst AND hFile <> 0 THEN
	bFailClose := TRUE;
	fbClose(sNetId := '', hFile := hFile, bExecute := TRUE, tTimeout := T#5S);
	eStep := E_MbLogWriterStep.CloseWait;
ELSE
	eStep := E_MbLogWriterStep.Idle;
END_IF
END_METHOD

METHOD PRIVATE NextLine : STRING(255)
VAR
	nAge, nIdx : UDINT;
END_VAR
// Entry with sequence number nCursor: nHead is the next write slot, newest is nHead-1
nAge := pLog^.nSeq - 1 - nCursor;
nIdx := (UINT_TO_UDINT(pLog^.nHead) + GVL_MbParam.MB_LOG_SIZE - 1 - nAge) MOD GVL_MbParam.MB_LOG_SIZE;
bLineIsEntry := TRUE;
NextLine := F_MbLogEntryToCsv(pLog^.aEntries[nIdx]);
END_METHOD

END_FUNCTION_BLOCK

// ---- POUs/Log/F_MbLogEntryToCsv.TcPOU
FUNCTION F_MbLogEntryToCsv : STRING(255)
VAR_INPUT
	stE  : ST_MbLogEntry;
END_VAR
VAR
	ft   : T_FILETIME;
	sOut : STRING(255);
END_VAR

ft.dwLowDateTime  := ULINT_TO_DWORD(stE.tTime);
ft.dwHighDateTime := ULINT_TO_DWORD(SHR(stE.tTime, 32));
sOut := SYSTEMTIME_TO_STRING(FILETIME_TO_SYSTEMTIME(ft));
sOut := CONCAT(sOut, ',');  sOut := CONCAT(sOut, stE.sName);
sOut := CONCAT(sOut, ',');  sOut := CONCAT(sOut, USINT_TO_STRING(stE.nUnitId));
sOut := CONCAT(sOut, ',');  sOut := CONCAT(sOut, TO_STRING(stE.eRegion));
sOut := CONCAT(sOut, ',');  sOut := CONCAT(sOut, UDINT_TO_STRING(stE.nAddr));
sOut := CONCAT(sOut, ',');  sOut := CONCAT(sOut, BYTE_TO_STRING(stE.nFc));
sOut := CONCAT(sOut, ',');  sOut := CONCAT(sOut, TO_STRING(stE.eOp));
sOut := CONCAT(sOut, ',');  sOut := CONCAT(sOut, TO_STRING(stE.eClass));
sOut := CONCAT(sOut, ',');  sOut := CONCAT(sOut, BYTE_TO_STRING(stE.nExcCode));
sOut := CONCAT(sOut, ',');  sOut := CONCAT(sOut, USINT_TO_STRING(stE.nRetries));
sOut := CONCAT(sOut, ',');  sOut := CONCAT(sOut, UDINT_TO_STRING(stE.nRepeat));
sOut := CONCAT(sOut, '$N');
F_MbLogEntryToCsv := sOut;

END_FUNCTION

// ---- POUs/Log/FB_MbLogExport.TcPOU
FUNCTION_BLOCK FB_MbLogExport
VAR_INPUT
	sPath    : STRING(255) := 'C:\ModbusExt\modbus_log.csv';   // Folder must exist
	bExecute : BOOL;                                           // Rising edge starts an export
	refLog   : REFERENCE TO ST_MbLog;
END_VAR
VAR_OUTPUT
	bBusy    : BOOL;
	bDone    : BOOL;
	bError   : BOOL;
	nErrId   : UDINT;
	nWritten : UINT;
END_VAR
VAR
	rtrig    : R_TRIG;
	fbOpen   : FB_FileOpen;
	fbPuts   : FB_FilePuts;
	fbClose  : FB_FileClose;
	hFile    : UINT;
	eStep    : USINT;
	nIdx     : UINT;
	nCount   : UINT;
	nStart   : UINT;
	sLine    : STRING(255);
END_VAR

rtrig(CLK := bExecute);
IF rtrig.Q AND eStep = 0 THEN
	IF NOT __ISVALIDREF(refLog) THEN
		bError := TRUE;
		bDone  := FALSE;
	ELSE
		bBusy    := TRUE;
		bDone    := FALSE;
		bError   := FALSE;
		nErrId   := 0;
		nWritten := 0;
		nCount   := MIN(refLog.nCount, GVL_MbParam.MB_LOG_SIZE);
		nStart   := (refLog.nHead + GVL_MbParam.MB_LOG_SIZE - nCount) MOD GVL_MbParam.MB_LOG_SIZE;   // Oldest entry
		nIdx     := 0;
		fbOpen(sNetId := '', sPathName := sPath, nMode := FOPEN_MODEWRITE OR FOPEN_MODETEXT,
		       ePath := PATH_GENERIC, bExecute := TRUE, tTimeout := T#5S);
		eStep := 1;
	END_IF
END_IF

CASE eStep OF
	1:  // Open
		fbOpen(bExecute := FALSE);
		IF NOT fbOpen.bBusy THEN
			IF fbOpen.bError THEN
				nErrId := fbOpen.nErrId;
				bError := TRUE;
				bBusy  := FALSE;
				eStep  := 0;
			ELSE
				hFile := fbOpen.hFile;
				sLine := 'TimeUTC,Name,Unit,Region,Address,FC,Op,Class,ExcCode,Retries,Repeat$N';
				fbPuts(sNetId := '', hFile := hFile, sLine := sLine, bExecute := TRUE, tTimeout := T#5S);
				eStep := 2;
			END_IF
		END_IF

	2:  // One line per ADS round trip
		fbPuts(bExecute := FALSE);
		IF NOT fbPuts.bBusy THEN
			IF fbPuts.bError THEN
				nErrId := fbPuts.nErrId;
				bError := TRUE;
				fbClose(sNetId := '', hFile := hFile, bExecute := TRUE, tTimeout := T#5S);
				eStep := 3;
			ELSIF nIdx < nCount THEN
				sLine := F_MbLogEntryToCsv(refLog.aEntries[(nStart + nIdx) MOD GVL_MbParam.MB_LOG_SIZE]);
				nIdx     := nIdx + 1;
				nWritten := nIdx;
				fbPuts(sNetId := '', hFile := hFile, sLine := sLine, bExecute := TRUE, tTimeout := T#5S);
			ELSE
				fbClose(sNetId := '', hFile := hFile, bExecute := TRUE, tTimeout := T#5S);
				eStep := 3;
			END_IF
		END_IF

	3:  // Close
		fbClose(bExecute := FALSE);
		IF NOT fbClose.bBusy THEN
			IF fbClose.bError AND NOT bError THEN
				nErrId := fbClose.nErrId;
				bError := TRUE;
			END_IF
			bDone := NOT bError;
			bBusy := FALSE;
			eStep := 0;
		END_IF
END_CASE

END_FUNCTION_BLOCK

// ---- POUs/Profiles/FB_Mb_CorrAll.TcPOU
(*@ModbusExt.Profile v1 - managed by ModbusExt Profile Editor. One point per line.*)
FUNCTION_BLOCK FB_Mb_CorrAll EXTENDS FB_ModbusDevice
VAR_INPUT
	Viscus : ST_MbPoint := (nAddr := 40001, eType := E_MbType.Int16, fRawMin := -16000, fRawMax := 16000, fEngMin := 0, fEngMax := 20);   // replace me
	Flow   : ST_MbPoint := (nAddr := 40002, eType := E_MbType.Int16);
	Temp   : ST_MbPoint := (nAddr := 40003, fGain := 1.8, fOffset := 32);
END_VAR

Register();
SUPER^();

METHOD PRIVATE Register
Profile(sModel := 'CorrAll');
AddPoint(Viscus, 'Viscus');
AddPoint(Flow, 'Flow');
AddPoint(Temp, 'Temp');
END_METHOD

END_FUNCTION_BLOCK

// ---- POUs/Transport/FB_MbTransportMock.TcPOU
FUNCTION_BLOCK FB_MbTransportMock IMPLEMENTS I_MbTransport
VAR_INPUT
	bReadyIn        : BOOL := TRUE;
	nDelayCycles    : UINT := 2;       // Poll() calls between Send and Done
	bForceTimeout   : BOOL;            // Answer Timeout
	bForceCrc       : BOOL;            // Answer Error / Crc
	bForceException : BOOL;            // Answer exception nForcedExc
	nForcedExc      : BYTE := 2;
	bExcOnRange     : BOOL;            // Exception 02 when a register read covers nExcOffset
	nExcOffset      : UINT;
	// Simulated device memory, 0-based. Inputs so test code can write them directly.
	aHolding        : ARRAY[0..999] OF WORD;
	aInput          : ARRAY[0..999] OF WORD;
	aCoils          : ARRAY[0..999] OF BOOL;
	aDiscrete       : ARRAY[0..999] OF BOOL;
END_VAR
VAR_OUTPUT
	nRequests       : UDINT;
	nOwner          : USINT;           // 0 = bus free
	nLastUnit       : USINT;
	nLastFc         : USINT;
	nLastOffset     : UINT;
	nLastQty        : UINT;            // Value field for FC5/6
END_VAR
VAR
	eState          : E_MbXferState;
	eErr            : E_MbErrorClass;
	aReq            : ARRAY[0..GVL_MbParam.MB_ADU_SIZE-1] OF BYTE;
	cbReq           : UINT;
	aResp           : ARRAY[0..GVL_MbParam.MB_ADU_SIZE-1] OF BYTE;
	cbResp          : UINT;
	nCountdown      : UINT;
END_VAR

METHOD Abort
VAR_INPUT
	nUnitId	: USINT;
END_VAR
IF nOwner = nUnitId THEN
	eState := E_MbXferState.Idle;
	cbResp := 0;
END_IF
END_METHOD

METHOD Acquire : BOOL
VAR_INPUT
	(* Caller's unit ID doubles as the owner key. TRUE = you hold the bus.*)
	nUnitId	: USINT;
END_VAR
IF nUnitId = 0 THEN
	Acquire := FALSE;
	RETURN;
END_IF
IF nOwner = 0 THEN
	nOwner := nUnitId;
END_IF
Acquire := (nOwner = nUnitId);
END_METHOD

PROPERTY bReady : BOOL
GET
bReady := bReadyIn;
END_GET
END_PROPERTY

PROPERTY cbResponsePdu : UINT
GET
cbResponsePdu := cbResp;
END_GET
END_PROPERTY

PROPERTY eLastError : E_MbErrorClass
GET
eLastError := eErr;
END_GET
END_PROPERTY

METHOD Poll : E_MbXferState
IF eState = E_MbXferState.Busy THEN
	IF nCountdown > 0 THEN
		nCountdown := nCountdown - 1;
	ELSE
		Respond();
	END_IF
END_IF
Poll := eState;
END_METHOD

PROPERTY pResponsePdu : POINTER TO BYTE
GET
pResponsePdu := ADR(aResp);
END_GET
END_PROPERTY

METHOD Release
VAR_INPUT
	nUnitId	: USINT;
END_VAR
IF nOwner = nUnitId THEN
	nOwner := 0;
	eState := E_MbXferState.Idle;
END_IF
END_METHOD

METHOD PRIVATE Respond
VAR
	nFc      : USINT;
	nOff     : UINT;
	nQty     : UINT;
	nByteCnt : UINT;
	i        : UINT;
	w        : WORD;
END_VAR
IF bForceTimeout THEN
	eState := E_MbXferState.Timeout;
	RETURN;
END_IF
IF bForceCrc THEN
	eState := E_MbXferState.Error;
	eErr   := E_MbErrorClass.Crc;
	RETURN;
END_IF

nFc  := BYTE_TO_USINT(aReq[0]);
nOff := nLastOffset;
nQty := nLastQty;

IF bForceException THEN
	SendException(nForcedExc);
	RETURN;
END_IF

CASE nFc OF
	GVL_MbConst.FC_READ_COILS, GVL_MbConst.FC_READ_DISCRETE:
		IF nQty < 1 OR nQty > GVL_MbConst.MAX_READ_COILS OR UINT_TO_UDINT(nOff) + nQty > 1000 THEN
			SendException(2);
			RETURN;
		END_IF
		nByteCnt := (nQty + 7) / 8;
		aResp[0] := aReq[0];
		aResp[1] := UINT_TO_BYTE(nByteCnt);
		F_MbMemSet(ADR(aResp[2]), 0, nByteCnt);
		FOR i := 0 TO nQty - 1 DO
			IF SEL(nFc = GVL_MbConst.FC_READ_COILS, aDiscrete[nOff + i], aCoils[nOff + i]) THEN
				aResp[2 + i / 8] := aResp[2 + i / 8] OR SHL(BYTE#1, i MOD 8);
			END_IF
		END_FOR
		cbResp := 2 + nByteCnt;

	GVL_MbConst.FC_READ_HOLDING, GVL_MbConst.FC_READ_INPUT:
		IF nQty < 1 OR nQty > GVL_MbConst.MAX_READ_REGS OR UINT_TO_UDINT(nOff) + nQty > 1000 THEN
			SendException(2);
			RETURN;
		END_IF
		IF bExcOnRange AND nExcOffset >= nOff AND nExcOffset < nOff + nQty THEN
			SendException(2);
			RETURN;
		END_IF
		aResp[0] := aReq[0];
		aResp[1] := UINT_TO_BYTE(2 * nQty);
		FOR i := 0 TO nQty - 1 DO
			IF nFc = GVL_MbConst.FC_READ_HOLDING THEN
				w := aHolding[nOff + i];
			ELSE
				w := aInput[nOff + i];
			END_IF
			aResp[2 + 2 * i] := WORD_TO_BYTE(SHR(w, 8));
			aResp[3 + 2 * i] := WORD_TO_BYTE(w);
		END_FOR
		cbResp := 2 + 2 * nQty;

	GVL_MbConst.FC_WRITE_COIL:
		IF nOff >= 1000 THEN
			SendException(2);
			RETURN;
		END_IF
		IF nQty = 16#FF00 THEN
			aCoils[nOff] := TRUE;
		ELSIF nQty = 0 THEN
			aCoils[nOff] := FALSE;
		ELSE
			SendException(3);
			RETURN;
		END_IF
		F_MbMemCpy(ADR(aResp), ADR(aReq), 5);
		cbResp := 5;

	GVL_MbConst.FC_WRITE_REGISTER:
		IF nOff >= 1000 THEN
			SendException(2);
			RETURN;
		END_IF
		aHolding[nOff] := UINT_TO_WORD(nQty);
		F_MbMemCpy(ADR(aResp), ADR(aReq), 5);
		cbResp := 5;

	GVL_MbConst.FC_WRITE_COILS:
		nByteCnt := (nQty + 7) / 8;
		IF nQty < 1 OR nQty > GVL_MbConst.MAX_WRITE_COILS OR UINT_TO_UDINT(nOff) + nQty > 1000 OR cbReq < 6 + nByteCnt THEN
			SendException(2);
			RETURN;
		END_IF
		FOR i := 0 TO nQty - 1 DO
			aCoils[nOff + i] := (aReq[6 + i / 8] AND SHL(BYTE#1, i MOD 8)) <> 0;
		END_FOR
		F_MbMemCpy(ADR(aResp), ADR(aReq), 5);
		cbResp := 5;

	GVL_MbConst.FC_WRITE_REGISTERS:
		IF nQty < 1 OR nQty > GVL_MbConst.MAX_WRITE_REGS OR UINT_TO_UDINT(nOff) + nQty > 1000 OR cbReq < 6 + 2 * nQty THEN
			SendException(2);
			RETURN;
		END_IF
		FOR i := 0 TO nQty - 1 DO
			aHolding[nOff + i] := SHL(BYTE_TO_WORD(aReq[6 + 2 * i]), 8) OR BYTE_TO_WORD(aReq[7 + 2 * i]);
		END_FOR
		F_MbMemCpy(ADR(aResp), ADR(aReq), 5);
		cbResp := 5;
ELSE
	SendException(1);
	RETURN;
END_CASE

eState := E_MbXferState.Done;
END_METHOD

METHOD Send : BOOL
VAR_INPUT
	nUnitId	: USINT;
	pPdu	: POINTER TO BYTE;
	cbPdu	: UINT;
	(* From F_MbExpectedResponseLength; RTU uses it to detect end of frame*)
	nExpectedPduLen	: UINT;
	tTimeout	: TIME;
END_VAR
Send := FALSE;
IF nOwner <> nUnitId OR NOT bReadyIn OR pPdu = 0 OR cbPdu < 1 OR cbPdu > GVL_MbParam.MB_ADU_SIZE THEN
	RETURN;
END_IF
F_MbMemCpy(ADR(aReq), pPdu, cbPdu);
cbReq      := cbPdu;
cbResp     := 0;
nCountdown := nDelayCycles;
eState     := E_MbXferState.Busy;
eErr       := E_MbErrorClass.None;
nLastUnit  := nUnitId;
nLastFc    := BYTE_TO_USINT(aReq[0]);
IF cbReq >= 5 THEN
	nLastOffset := SHL(BYTE_TO_UINT(aReq[1]), 8) + BYTE_TO_UINT(aReq[2]);
	nLastQty    := SHL(BYTE_TO_UINT(aReq[3]), 8) + BYTE_TO_UINT(aReq[4]);
END_IF
nRequests := nRequests + 1;
Send := TRUE;
END_METHOD

METHOD PRIVATE SendException
VAR_INPUT
	nCode : BYTE;
END_VAR
aResp[0] := aReq[0] OR GVL_MbConst.EXC_FLAG;
aResp[1] := nCode;
cbResp   := 2;
eState   := E_MbXferState.Done;   // An exception is a valid frame; the device's parser classifies it
END_METHOD

END_FUNCTION_BLOCK

// ---- POUs/Transport/FB_MbTransportRtu.TcPOU
FUNCTION_BLOCK FB_MbTransportRtu IMPLEMENTS I_MbTransport
VAR_INPUT
	eMode       : ComSerialLineMode_t := SERIALLINEMODE_EL6_22B;   // Tc2_SerialCom line mode for the linked terminal
	pComIn      : POINTER TO ARRAY[0..65] OF BYTE;   // ADR() of the linked input struct, e.g. EL6inData22B;                                 // ADR() of the linked input struct, e.g. EL6inData22B
	pComOut     : POINTER TO ARRAY[0..65] OF BYTE;   // ADR() of the linked output struct, e.g. EL6outData22B                                 // ADR() of the linked output struct, e.g. EL6outData22B
	nSizeComIn  : UINT;                                  // SIZEOF() of the input struct
	tInterFrame : TIME := T#10MS;                        // Bus idle enforced between transactions
	tGap        : TIME := T#20MS;                        // Silence that ends a frame of unexpected length
	bEnable     : BOOL := TRUE;
END_VAR
VAR_OUTPUT
	bLineOk     : BOOL;
	eLineErr    : ComError_t;
	nOwner      : USINT;
	nTxCount    : UDINT;
	nRxCount    : UDINT;
	nCrcErrors  : UDINT;
END_VAR
VAR
	fbLine      : SerialLineControl;
	TxBuffer    : ComBuffer;
	RxBuffer    : ComBuffer;
	fbSendByte  : SendByte;
	fbRecvByte  : ReceiveByte;
	fbSysTime   : GETSYSTEMTIME;
	tNow        : ULINT;

	eState      : E_MbXferState;
	eErr        : E_MbErrorClass;
	nUnitReq    : USINT;
	nExpectedPdu : UINT;
	tTimeoutTicks : ULINT;
	tDeadline   : ULINT;
	tNextTxAllowed : ULINT;
	tLastByte   : ULINT;
	bTxStarted  : BOOL;

	aTx         : ARRAY[0..GVL_MbParam.MB_ADU_SIZE-1] OF BYTE;   // unit id + PDU + CRC
	cbTx        : UINT;
	nTxSent     : UINT;
	aRx         : ARRAY[0..GVL_MbParam.MB_ADU_SIZE-1] OF BYTE;
	cbRx        : UINT;
	aResp       : ARRAY[0..GVL_MbParam.MB_ADU_SIZE-1] OF BYTE;   // PDU handed to the device
	cbResp      : UINT;
END_VAR

fbSysTime();
tNow := SHL(DWORD_TO_ULINT(fbSysTime.timeHiDW), 32) + DWORD_TO_ULINT(fbSysTime.timeLoDW);

IF pComIn = 0 OR pComOut = 0 OR nSizeComIn = 0 THEN
	bLineOk := FALSE;
	RETURN;
END_IF

// Moves up to 22 bytes per cycle each way between the terminal image and the ComBuffers
fbLine(Mode := eMode, pComIn := pComIn, pComOut := pComOut, SizeComIn := UINT_TO_INT(nSizeComIn),
       TxBuffer := TxBuffer, RxBuffer := RxBuffer);
bLineOk  := bEnable AND NOT fbLine.Error;
eLineErr := fbLine.ErrorID;

IF eState <> E_MbXferState.Busy THEN
	Drain();                              // Keep the receive buffer empty between transactions
	RETURN;
END_IF
IF fbLine.Error THEN
	eState := E_MbXferState.Error;
	eErr   := E_MbErrorClass.Transport;
	RETURN;
END_IF

// 1. Respect the inter-frame gap, then hand the request to the line
IF NOT bTxStarted THEN
	IF tNow < tNextTxAllowed THEN
		RETURN;
	END_IF
	Drain();
	bTxStarted := TRUE;
	tDeadline  := tNow + tTimeoutTicks;   // Timeout counts from the real transmission start
	tLastByte  := tNow;
END_IF
WHILE nTxSent < cbTx DO
	fbSendByte(SendByte := aTx[nTxSent], TxBuffer := TxBuffer);
	IF fbSendByte.Busy THEN
		EXIT;                             // Buffer full; continue next cycle
	END_IF
	nTxSent := nTxSent + 1;
END_WHILE
IF nTxSent < cbTx THEN
	RETURN;
END_IF

// 2. Collect response bytes
Collect();

// 3. End of frame: by expected length, by exception frame, or by silence
IF cbRx >= 2 AND_THEN (aRx[1] AND GVL_MbConst.EXC_FLAG) <> 0 THEN
	IF cbRx >= 5 THEN
		Complete(5);
	END_IF
ELSIF nExpectedPdu > 0 AND cbRx >= 1 + nExpectedPdu + 2 THEN
	Complete(1 + nExpectedPdu + 2);
ELSIF cbRx >= 5 AND tNow - tLastByte >= F_MbTimeToFt(tGap) THEN
	Complete(cbRx);                       // Unexpected length; the CRC decides
END_IF

IF eState = E_MbXferState.Busy AND tNow >= tDeadline THEN
	eState         := E_MbXferState.Timeout;
	tNextTxAllowed := tNow + F_MbTimeToFt(tInterFrame);
END_IF

METHOD Abort
VAR_INPUT
	nUnitId	: USINT;
END_VAR
IF nOwner = nUnitId THEN
	eState         := E_MbXferState.Idle;
	cbRx           := 0;
	cbResp         := 0;
	tNextTxAllowed := tNow + F_MbTimeToFt(tInterFrame);   // Let a late answer die on the wire
END_IF
END_METHOD

METHOD Acquire : BOOL
VAR_INPUT
	(* Caller's unit ID doubles as the owner key. TRUE = you hold the bus.*)
	nUnitId	: USINT;
END_VAR
IF nUnitId = 0 THEN
	Acquire := FALSE;                     // Broadcast has no response; not supported
	RETURN;
END_IF
IF nOwner = 0 THEN
	nOwner := nUnitId;
END_IF
Acquire := (nOwner = nUnitId);
END_METHOD

PROPERTY bReady : BOOL
GET
bReady := bLineOk;
END_GET
END_PROPERTY

PROPERTY cbResponsePdu : UINT
GET
cbResponsePdu := cbResp;
END_GET
END_PROPERTY

METHOD PRIVATE Collect
WHILE cbRx < GVL_MbParam.MB_ADU_SIZE DO
	fbRecvByte(RxBuffer := RxBuffer);
	IF NOT fbRecvByte.ByteReceived THEN
		EXIT;
	END_IF
	aRx[cbRx] := fbRecvByte.ReceivedByte;
	cbRx      := cbRx + 1;
	tLastByte := tNow;
END_WHILE
END_METHOD

METHOD PRIVATE Complete
VAR_INPUT
	n    : UINT;   // Frame length including unit id and CRC
END_VAR
VAR
	wCrc : WORD;
END_VAR
tNextTxAllowed := tNow + F_MbTimeToFt(tInterFrame);
IF aRx[0] <> USINT_TO_BYTE(nUnitReq) THEN
	eState := E_MbXferState.Error;
	eErr   := E_MbErrorClass.Malformed;      // Answer from the wrong unit
	RETURN;
END_IF
wCrc := F_MbCrc16(ADR(aRx), n - 2);
IF aRx[n - 2] <> WORD_TO_BYTE(wCrc) OR aRx[n - 1] <> WORD_TO_BYTE(SHR(wCrc, 8)) THEN
	nCrcErrors := nCrcErrors + 1;
	eState     := E_MbXferState.Error;
	eErr       := E_MbErrorClass.Crc;
	RETURN;
END_IF
cbResp := n - 3;
F_MbMemCpy(ADR(aResp), ADR(aRx[1]), cbResp);
eState   := E_MbXferState.Done;
nRxCount := nRxCount + 1;
END_METHOD

METHOD PRIVATE Drain
VAR
	n : UINT;
END_VAR
// Discard whatever is sitting in the receive buffer (bounded loop)
FOR n := 1 TO 300 DO
	fbRecvByte(RxBuffer := RxBuffer);
	IF NOT fbRecvByte.ByteReceived THEN
		EXIT;
	END_IF
END_FOR
END_METHOD

PROPERTY eLastError : E_MbErrorClass
GET
eLastError := eErr;
END_GET
END_PROPERTY

METHOD Poll : E_MbXferState
Poll := eState;
END_METHOD

PROPERTY pResponsePdu : POINTER TO BYTE
GET
pResponsePdu := ADR(aResp);
END_GET
END_PROPERTY

METHOD Release
VAR_INPUT
	nUnitId	: USINT;
END_VAR
IF nOwner = nUnitId THEN
	nOwner := 0;
	IF eState <> E_MbXferState.Busy THEN
		eState := E_MbXferState.Idle;
	END_IF
END_IF
END_METHOD

METHOD Send : BOOL
VAR_INPUT
	nUnitId         : USINT;
	pPdu            : POINTER TO BYTE;
	cbPdu           : UINT;
	nExpectedPduLen : UINT;
	tTimeout        : TIME;
END_VAR
VAR
	wCrc            : WORD;
END_VAR
Send := FALSE;
IF nOwner <> nUnitId OR NOT bLineOk OR eState = E_MbXferState.Busy
   OR pPdu = 0 OR cbPdu < 1 OR cbPdu > GVL_MbParam.MB_ADU_SIZE - 3 THEN
	RETURN;
END_IF

aTx[0] := USINT_TO_BYTE(nUnitId);
F_MbMemCpy(ADR(aTx[1]), pPdu, cbPdu);
wCrc := F_MbCrc16(ADR(aTx), cbPdu + 1);
aTx[cbPdu + 1] := WORD_TO_BYTE(wCrc);              // Low byte first on the wire
aTx[cbPdu + 2] := WORD_TO_BYTE(SHR(wCrc, 8));
cbTx := cbPdu + 3;

nTxSent       := 0;
bTxStarted    := FALSE;
cbRx          := 0;
cbResp        := 0;
nUnitReq      := nUnitId;
nExpectedPdu  := nExpectedPduLen;
tTimeoutTicks := F_MbTimeToFt(tTimeout);
eErr          := E_MbErrorClass.None;
eState        := E_MbXferState.Busy;
nTxCount      := nTxCount + 1;
Send := TRUE;
END_METHOD

END_FUNCTION_BLOCK

// ---- POUs/Transport/FB_MbTransportTcp.TcPOU
FUNCTION_BLOCK FB_MbTransportTcp IMPLEMENTS I_MbTransport
VAR_INPUT
	sHost             : STRING(15) := '127.0.0.1';
	nPort             : UINT := 502;
	bEnable           : BOOL := TRUE;
	tConnectTimeout   : TIME := T#5S;
	tReconnectBackoff : TIME := T#2S;
END_VAR
VAR_OUTPUT
	bConnected        : BOOL;
	nConnects         : UDINT;
	nErrorId          : UDINT;        // Last TF6310 error code
	nOwner            : USINT;        // 0 = bus free
	nTxCount          : UDINT;
	nRxCount          : UDINT;
END_VAR
VAR
	eConn             : E_MbTcpConn;
	fbCloseAll        : FB_SocketCloseAll;
	fbConnect         : FB_SocketConnect;
	fbSend            : FB_SocketSend;
	fbReceive         : FB_SocketReceive;
	fbClose           : FB_SocketClose;
	hSocket           : T_HSOCKET;
	fbSysTime         : GETSYSTEMTIME;
	tNow              : ULINT;
	tBackoffUntil     : ULINT;

	eState            : E_MbXferState;
	eErr              : E_MbErrorClass;
	nTid              : UINT;
	nUnitReq          : USINT;
	tDeadline         : ULINT;
	bSendPhase        : BOOL;         // fbSend job outstanding
	bRecvArmed        : BOOL;         // fbReceive job outstanding
	nRxArmOffset      : UINT;         // Where the armed receive writes

	aTx               : ARRAY[0..GVL_MbParam.MB_ADU_SIZE-1] OF BYTE;   // MBAP + PDU
	cbTx              : UINT;
	aRx               : ARRAY[0..GVL_MbParam.MB_ADU_SIZE-1] OF BYTE;   // Reassembly buffer
	cbRx              : UINT;
	aResp             : ARRAY[0..GVL_MbParam.MB_ADU_SIZE-1] OF BYTE;   // PDU handed to the device
	cbResp            : UINT;
END_VAR

fbSysTime();
tNow := SHL(DWORD_TO_ULINT(fbSysTime.timeHiDW), 32) + DWORD_TO_ULINT(fbSysTime.timeLoDW);

// ---- Pump outstanding socket jobs (in every state, so nothing is left dangling) ----
IF bSendPhase THEN
	fbSend(bExecute := FALSE);
	IF NOT fbSend.bBusy THEN
		bSendPhase := FALSE;
		IF fbSend.bError THEN
			nErrorId := fbSend.nErrId;
			IF eConn = E_MbTcpConn.Connected THEN
				Disconnect();
			END_IF
		END_IF
	END_IF
END_IF
IF bRecvArmed THEN
	fbReceive(bExecute := FALSE);
	IF NOT fbReceive.bBusy THEN
		bRecvArmed := FALSE;
		IF fbReceive.bError THEN
			nErrorId := fbReceive.nErrId;
			IF eConn = E_MbTcpConn.Connected THEN
				Disconnect();
			END_IF
		ELSIF fbReceive.nRecBytes > 0 AND eConn = E_MbTcpConn.Connected THEN
			OnBytes(nRxArmOffset, UDINT_TO_UINT(fbReceive.nRecBytes));
		END_IF
	END_IF
END_IF

// ---- Connection management ----
CASE eConn OF
	E_MbTcpConn.Init:
		fbCloseAll(sSrvNetId := '', bExecute := TRUE, tTimeout := T#5S);   // Drop handles leaked by a previous run
		eConn := E_MbTcpConn.CloseAllWait;

	E_MbTcpConn.CloseAllWait:
		fbCloseAll(bExecute := FALSE);
		IF NOT fbCloseAll.bBusy THEN
			eConn := E_MbTcpConn.Disconnected;
		END_IF

	E_MbTcpConn.Disconnected:
		bConnected := FALSE;
		IF bEnable AND tNow >= tBackoffUntil THEN
			fbConnect(sSrvNetId := '', sRemoteHost := sHost, nRemotePort := nPort, bExecute := TRUE, tTimeout := tConnectTimeout);
			eConn := E_MbTcpConn.Connecting;
		END_IF

	E_MbTcpConn.Connecting:
		fbConnect(bExecute := FALSE);
		IF NOT fbConnect.bBusy THEN
			IF fbConnect.bError THEN
				nErrorId      := fbConnect.nErrId;
				tBackoffUntil := tNow + F_MbTimeToFt(tReconnectBackoff);
				eConn         := E_MbTcpConn.Disconnected;
			ELSE
				hSocket    := fbConnect.hSocket;
				bConnected := TRUE;
				nConnects  := nConnects + 1;
				eConn      := E_MbTcpConn.Connected;
			END_IF
		END_IF

	E_MbTcpConn.Connected:
		IF NOT bEnable THEN
			Disconnect();
		ELSE
			PumpTransaction();
		END_IF

	E_MbTcpConn.Closing:
		fbClose(sSrvNetId := '', hSocket := hSocket, bExecute := TRUE, tTimeout := T#5S);
		eConn := E_MbTcpConn.ClosingWait;

	E_MbTcpConn.ClosingWait:
		fbClose(bExecute := FALSE);
		IF NOT fbClose.bBusy THEN
			bConnected    := FALSE;
			tBackoffUntil := tNow + F_MbTimeToFt(tReconnectBackoff);
			eConn         := E_MbTcpConn.Disconnected;
		END_IF
END_CASE

METHOD Abort
VAR_INPUT
	nUnitId	: USINT;
END_VAR
IF nOwner = nUnitId THEN
	eState := E_MbXferState.Idle;
	cbRx   := 0;
	cbResp := 0;
END_IF
END_METHOD

METHOD Acquire : BOOL
VAR_INPUT
	(* Caller's unit ID doubles as the owner key. TRUE = you hold the bus.*)
	nUnitId	: USINT;
END_VAR
IF nUnitId = 0 THEN
	Acquire := FALSE;
	RETURN;
END_IF
IF nOwner = 0 THEN
	nOwner := nUnitId;
END_IF
Acquire := (nOwner = nUnitId);
END_METHOD

METHOD PRIVATE ArmReceive
IF cbRx >= GVL_MbParam.MB_ADU_SIZE THEN     // Buffer full without a frame: garbage
	cbRx   := 0;
	eState := E_MbXferState.Error;
	eErr   := E_MbErrorClass.Malformed;
	RETURN;
END_IF
nRxArmOffset := cbRx;
fbReceive(sSrvNetId := '', hSocket := hSocket, cbLen := GVL_MbParam.MB_ADU_SIZE - cbRx,
          pDest := ADR(aRx[cbRx]), bExecute := TRUE, tTimeout := T#5S);
bRecvArmed := TRUE;
END_METHOD

PROPERTY bReady : BOOL
GET
bReady := bConnected;
END_GET
END_PROPERTY

PROPERTY cbResponsePdu : UINT
GET
cbResponsePdu := cbResp;
END_GET
END_PROPERTY

METHOD PRIVATE Disconnect
IF eState = E_MbXferState.Busy THEN
	eState := E_MbXferState.Error;
	eErr   := E_MbErrorClass.Transport;
END_IF
cbRx  := 0;
eConn := E_MbTcpConn.Closing;
END_METHOD

PROPERTY eLastError : E_MbErrorClass
GET
eLastError := eErr;
END_GET
END_PROPERTY

METHOD PRIVATE OnBytes
VAR_INPUT
	nOffset : UINT;   // Where the receive wrote
	n       : UINT;
END_VAR
VAR
	nLen    : UINT;   // MBAP length field: unit id + PDU
	nFrame  : UINT;
	nTidRx  : UINT;
	nPid    : UINT;
END_VAR
// Realign if the buffer was reset while the receive was in flight
IF nOffset <> cbRx THEN
	F_MbMemCpy(ADR(aRx[cbRx]), ADR(aRx[nOffset]), n);
END_IF
cbRx := cbRx + n;

// Extract complete MBAP frames
WHILE cbRx >= 7 DO
	nLen := SHL(BYTE_TO_UINT(aRx[4]), 8) + BYTE_TO_UINT(aRx[5]);
	IF nLen < 2 OR nLen > GVL_MbParam.MB_ADU_SIZE - 6 THEN
		cbRx   := 0;
		eState := E_MbXferState.Error;
		eErr   := E_MbErrorClass.Malformed;
		RETURN;
	END_IF
	nFrame := 6 + nLen;
	IF cbRx < nFrame THEN
		RETURN;                                   // Wait for the rest
	END_IF
	nTidRx := SHL(BYTE_TO_UINT(aRx[0]), 8) + BYTE_TO_UINT(aRx[1]);
	nPid   := SHL(BYTE_TO_UINT(aRx[2]), 8) + BYTE_TO_UINT(aRx[3]);
	IF nPid = 0 AND nTidRx = nTid AND eState = E_MbXferState.Busy THEN
		cbResp := nLen - 1;
		F_MbMemCpy(ADR(aResp), ADR(aRx[7]), cbResp);
		eState   := E_MbXferState.Done;
		nRxCount := nRxCount + 1;
	END_IF                                        // Otherwise stale: drop it
	IF cbRx > nFrame THEN
		F_MbMemCpy(ADR(aRx), ADR(aRx[nFrame]), cbRx - nFrame);
	END_IF
	cbRx := cbRx - nFrame;
END_WHILE
END_METHOD

METHOD Poll : E_MbXferState
Poll := eState;   // The body does the work
END_METHOD

PROPERTY pResponsePdu : POINTER TO BYTE
GET
pResponsePdu := ADR(aResp);
END_GET
END_PROPERTY

METHOD PRIVATE PumpTransaction
IF eState <> E_MbXferState.Busy THEN
	RETURN;
END_IF
IF tNow >= tDeadline THEN
	eState := E_MbXferState.Timeout;
	RETURN;
END_IF
IF NOT bSendPhase AND NOT bRecvArmed THEN
	ArmReceive();
END_IF
END_METHOD

METHOD Release
VAR_INPUT
	nUnitId	: USINT;
END_VAR
IF nOwner = nUnitId THEN
	nOwner := 0;
	IF eState <> E_MbXferState.Busy THEN
		eState := E_MbXferState.Idle;
	END_IF
END_IF
END_METHOD

METHOD Send : BOOL
VAR_INPUT
	nUnitId	: USINT;
	pPdu	: POINTER TO BYTE;
	cbPdu	: UINT;
	(* From F_MbExpectedResponseLength; RTU uses it to detect end of frame*)
	nExpectedPduLen	: UINT;
	tTimeout	: TIME;
END_VAR
Send := FALSE;
IF nOwner <> nUnitId OR NOT bConnected OR eState = E_MbXferState.Busy OR bSendPhase
   OR pPdu = 0 OR cbPdu < 1 OR cbPdu > GVL_MbParam.MB_ADU_SIZE - 7 THEN
	RETURN;
END_IF

// MBAP: transaction id, protocol id 0, length (unit id + PDU), unit id
nTid := nTid + 1;
IF nTid = 0 THEN
	nTid := 1;
END_IF
aTx[0] := UINT_TO_BYTE(SHR(nTid, 8));
aTx[1] := UINT_TO_BYTE(nTid);
aTx[2] := 0;
aTx[3] := 0;
aTx[4] := UINT_TO_BYTE(SHR(cbPdu + 1, 8));
aTx[5] := UINT_TO_BYTE(cbPdu + 1);
aTx[6] := USINT_TO_BYTE(nUnitId);
F_MbMemCpy(ADR(aTx[7]), pPdu, cbPdu);
cbTx := 7 + cbPdu;

cbRx      := 0;                       // Anything stale is dropped; a late frame fails the TID check anyway
cbResp    := 0;
nUnitReq  := nUnitId;
eErr      := E_MbErrorClass.None;
tDeadline := tNow + F_MbTimeToFt(tTimeout);
fbSend(sSrvNetId := '', hSocket := hSocket, cbLen := cbTx, pSrc := ADR(aTx), bExecute := TRUE, tTimeout := T#5S);
bSendPhase := TRUE;
eState     := E_MbXferState.Busy;
nTxCount   := nTxCount + 1;
Send := TRUE;
END_METHOD

END_FUNCTION_BLOCK
